gfCNCPoint5[27571] = {X 492.8890, Y 40.6660, Z -8.0000, A 0.000, B 0.000, C 0.000 }
gfCNCPoint5[27572] = {X 492.8890, Y 35.0338, Z -8.0000, A 0.000, B 0.000, C 0.000 }
gfCNCPoint5[27573] = {X 491.0677, Y 35.0338, Z -8.0000, A 0.000, B 0.000, C 0.000 }
gfCNCPoint5[27574] = {X 487.0438, Y 42.8699, Z -8.0000, A 0.000, B 0.000, C 0.000 }
gfCNCPoint5[27575] = {X 487.1809, Y 43.5111, Z -8.0000, A 0.000, B 0.000, C 0.000 }
gfCNCPoint5[27576] = {X 487.2308, Y 44.1648, Z -8.0000, A 0.000, B 0.000, C 0.000 }
gfCNCPoint5[27577] = {X 487.2310, Y 45.0000, Z -8.0000, A 0.000, B 0.000, C 0.000 }
gfCNCPoint5[27578] = {X 487.1749, Y 45.7380, Z -8.0000, A 0.000, B 0.000, C 0.000 }
gfCNCPoint5[27579] = {X 487.0078, Y 46.4590, Z -8.0000, A 0.000, B 0.000, C 0.000 }
gfCNCPoint5[27580] = {X 486.5939, Y 47.4110, Z -8.0000, A 0.000, B 0.000, C 0.000 }
gfCNCPoint5[27581] = {X 485.9879, Y 48.2538, Z -8.0000, A 0.000, B 0.000, C 0.000 }
gfCNCPoint5[27582] = {X 485.2175, Y 48.9494, Z -8.0000, A 0.000, B 0.000, C 0.000 }
gfCNCPoint5[27583] = {X 484.3173, Y 49.4663, Z -8.0000, A 0.000, B 0.000, C 0.000 }
gfCNCPoint5[27584] = {X 483.3557, Y 49.7755, Z -8.0000, A 0.000, B 0.000, C 0.000 }
gfCNCPoint5[27585] = {X 482.3510, Y 49.8800, Z -8.0000, A 0.000, B 0.000, C 0.000 }
gfCNCPoint5[27586] = {X 480.2695, Y 49.8800, Z -8.0000, A 0.000, B 0.000, C 0.000 }
gfCNCPoint5[27587] = {X 480.2695, Y 49.4000, Z -8.0000, A 0.000, B 0.000, C 0.000 }
gfCNCPoint5[27588] = {X 475.7650, Y 49.4000, Z -8.0000, A 0.000, B 0.000, C 0.000 }
gfCNCPoint5[27589] = {X 474.7859, Y 49.2897, Z -8.0000, A 0.000, B 0.000, C 0.000 }
gfCNCPoint5[27590] = {X 473.8559, Y 48.9643, Z -8.0000, A 0.000, B 0.000, C 0.000 }
gfCNCPoint5[27591] = {X 473.0216, Y 48.4401, Z -8.0000, A 0.000, B 0.000, C 0.000 }
gfCNCPoint5[27592] = {X 472.3249, Y 47.7434, Z -8.0000, A 0.000, B 0.000, C 0.000 }
gfCNCPoint5[27593] = {X 471.8007, Y 46.9091, Z -8.0000, A 0.000, B 0.000, C 0.000 }
gfCNCPoint5[27594] = {X 471.4753, Y 45.9791, Z -8.0000, A 0.000, B 0.000, C 0.000 }
gfCNCPoint5[27595] = {X 471.3650, Y 45.0000, Z -8.0000, A 0.000, B 0.000, C 0.000 }
gfCNCPoint5[27596] = {X 471.3654, Y 44.1483, Z -8.0000, A 0.000, B 0.000, C 0.000 }
gfCNCPoint5[27597] = {X 471.4638, Y 43.2816, Z -8.0000, A 0.000, B 0.000, C 0.000 }
gfCNCPoint5[27598] = {X 471.7311, Y 42.4514, Z -8.0000, A 0.000, B 0.000, C 0.000 }
gfCNCPoint5[27599] = {X 472.1570, Y 41.6903, Z -8.0000, A 0.000, B 0.000, C 0.000 }
gfCNCPoint5[27600] = {X 472.7247, Y 41.0281, Z -8.0000, A 0.000, B 0.000, C 0.000 }
gfCNCPoint5[27601] = {X 473.4118, Y 40.4909, Z -8.0000, A 0.000, B 0.000, C 0.000 }
gfCNCPoint5[27602] = {X 474.1914, Y 40.0998, Z -8.0000, A 0.000, B 0.000, C 0.000 }
gfCNCPoint5[27603] = {X 478.1276, Y 32.3951, Z -8.0000, A 0.000, B 0.000, C 0.000 }
gfCNCPoint5[27604] = {X 476.8700, Y 31.5216, Z -8.0000, A 0.000, B 0.000, C 0.000 }
gfCNCPoint5[27605] = {X 475.7393, Y 30.4892, Z -8.0000, A 0.000, B 0.000, C 0.000 }
gfCNCPoint5[27606] = {X 474.7552, Y 29.3160, Z -8.0000, A 0.000, B 0.000, C 0.000 }
gfCNCPoint5[27607] = {X 473.9353, Y 28.0229, Z -8.0000, A 0.000, B 0.000, C 0.000 }
gfCNCPoint5[27608] = {X 473.2938, Y 26.6325, Z -8.0000, A 0.000, B 0.000, C 0.000 }
gfCNCPoint5[27609] = {X 472.8423, Y 25.1695, Z -8.0000, A 0.000, B 0.000, C 0.000 }
gfCNCPoint5[27610] = {X 472.5272, Y 23.4783, Z -8.0000, A 0.000, B 0.000, C 0.000 }
gfCNCPoint5[27611] = {X 472.3864, Y 21.7639, Z -8.0000, A 0.000, B 0.000, C 0.000 }
gfCNCPoint5[27612] = {X 472.4213, Y 20.0441, Z -8.0000, A 0.000, B 0.000, C 0.000 }
gfCNCPoint5[27613] = {X 472.6315, Y 18.3368, Z -8.0000, A 0.000, B 0.000, C 0.000 }
gfCNCPoint5[27614] = {X 473.0148, Y 16.6598, Z -8.0000, A 0.000, B 0.000, C 0.000 }
gfCNCPoint5[27615] = {X 473.5615, Y 15.1345, Z -8.0000, A 0.000, B 0.000, C 0.000 }
gfCNCPoint5[27616] = {X 474.3101, Y 13.6975, Z -8.0000, A 0.000, B 0.000, C 0.000 }
gfCNCPoint5[27617] = {X 475.2468, Y 12.3754, Z -8.0000, A 0.000, B 0.000, C 0.000 }
gfCNCPoint5[27618] = {X 476.3541, Y 11.1925, Z -8.0000, A 0.000, B 0.000, C 0.000 }
gfCNCPoint5[27619] = {X 477.6116, Y 10.1708, Z -8.0000, A 0.000, B 0.000, C 0.000 }
gfCNCPoint5[27620] = {X 478.9962, Y 9.3291, Z -8.0000, A 0.000, B 0.000, C 0.000 }
gfCNCPoint5[27621] = {X 480.4821, Y 8.6830, Z -8.0000, A 0.000, B 0.000, C 0.000 }
gfCNCPoint5[27622] = {X 482.0419, Y 8.2445, Z -8.0000, A 0.000, B 0.000, C 0.000 }
gfCNCPoint5[27623] = {X 484.1468, Y 7.9165, Z -8.0000, A 0.000, B 0.000, C 0.000 }
gfCNCPoint5[27624] = {X 486.2739, Y 7.8014, Z -8.0000, A 0.000, B 0.000, C 0.000 }
gfCNCPoint5[27625] = {X 486.9707, Y 7.7892, Z -8.0000, A 0.000, B 0.000, C 0.000 }
gfCNCPoint5[27626] = {X 502.2084, Y 7.7892, Z -8.0000, A 0.000, B 0.000, C 0.000 }
gfCNCPoint5[27627] = {X 502.7400, Y 7.7934, Z -8.0000, A 0.000, B 0.000, C 0.000 }
gfCNCPoint5[27628] = {X 503.7096, Y 7.9098, Z -8.0000, A 0.000, B 0.000, C 0.000 }
gfCNCPoint5[27629] = {X 504.6294, Y 8.2380, Z -8.0000, A 0.000, B 0.000, C 0.000 }
gfCNCPoint5[27630] = {X 505.4536, Y 8.7617, Z -8.0000, A 0.000, B 0.000, C 0.000 }
gfCNCPoint5[27631] = {X 506.1415, Y 9.4549, Z -8.0000, A 0.000, B 0.000, C 0.000 }
gfCNCPoint5[27632] = {X 506.6587, Y 10.2832, Z -8.0000, A 0.000, B 0.000, C 0.000 }
gfCNCPoint5[27633] = {X 506.9797, Y 11.2055, Z -8.0000, A 0.000, B 0.000, C 0.000 }
gfCNCPoint5[27634] = {X 507.0885, Y 12.1759, Z -8.0000, A 0.000, B 0.000, C 0.000 }
gfCNCPoint5[27635] = {X 507.0883, Y 13.0233, Z -8.0000, A 0.000, B 0.000, C 0.000 }
gfCNCPoint5[27636] = {X 506.9800, Y 13.9491, Z -8.0000, A 0.000, B 0.000, C 0.000 }
gfCNCPoint5[27637] = {X 506.6792, Y 14.8313, Z -8.0000, A 0.000, B 0.000, C 0.000 }
gfCNCPoint5[27638] = {X 506.1993, Y 15.6303, Z -8.0000, A 0.000, B 0.000, C 0.000 }
gfCNCPoint5[27639] = {X 505.5618, Y 16.3103, Z -8.0000, A 0.000, B 0.000, C 0.000 }
gfCNCPoint5[27640] = {X 505.5624, Y 40.8770, Z -8.0000, A 0.000, B 0.000, C 0.000 }
gfCNCPoint5[27641] = {X 506.2064, Y 41.5660, Z -8.0000, A 0.000, B 0.000, C 0.000 }
gfCNCPoint5[27642] = {X 506.6888, Y 42.3765, Z -8.0000, A 0.000, B 0.000, C 0.000 }
gfCNCPoint5[27643] = {X 506.9874, Y 43.2711, Z -8.0000, A 0.000, B 0.000, C 0.000 }
gfCNCPoint5[27644] = {X 507.0885, Y 44.2089, Z -8.0000, A 0.000, B 0.000, C 0.000 }
gfCNCPoint5[27645] = {X 507.0885, Y 45.0000, Z -8.0000, A 0.000, B 0.000, C 0.000 }
gfCNCPoint5[27646] = {X 506.9782, Y 45.9791, Z -8.0000, A 0.000, B 0.000, C 0.000 }
gfCNCPoint5[27647] = {X 506.6528, Y 46.9091, Z -8.0000, A 0.000, B 0.000, C 0.000 }
gfCNCPoint5[27648] = {X 506.1285, Y 47.7434, Z -8.0000, A 0.000, B 0.000, C 0.000 }
gfCNCPoint5[27649] = {X 505.4318, Y 48.4401, Z -8.0000, A 0.000, B 0.000, C 0.000 }
gfCNCPoint5[27650] = {X 504.5976, Y 48.9643, Z -8.0000, A 0.000, B 0.000, C 0.000 }
gfCNCPoint5[27651] = {X 503.6676, Y 49.2897, Z -8.0000, A 0.000, B 0.000, C 0.000 }
gfCNCPoint5[27652] = {X 502.6885, Y 49.4000, Z -8.0000, A 0.000, B 0.000, C 0.000 }
gfCNCPoint5[27653] = {X 496.2450, Y 49.4000, Z -8.0000, A 0.000, B 0.000, C 0.000 }
gfCNCPoint5[27654] = {X 495.2659, Y 49.2897, Z -8.0000, A 0.000, B 0.000, C 0.000 }
gfCNCPoint5[27655] = {X 494.3359, Y 48.9643, Z -8.0000, A 0.000, B 0.000, C 0.000 }
gfCNCPoint5[27656] = {X 493.5017, Y 48.4401, Z -8.0000, A 0.000, B 0.000, C 0.000 }
gfCNCPoint5[27657] = {X 492.8050, Y 47.7433, Z -8.0000, A 0.000, B 0.000, C 0.000 }
gfCNCPoint5[27658] = {X 492.2808, Y 46.9091, Z -8.0000, A 0.000, B 0.000, C 0.000 }
gfCNCPoint5[27659] = {X 491.9553, Y 45.9791, Z -8.0000, A 0.000, B 0.000, C 0.000 }
gfCNCPoint5[27660] = {X 491.8450, Y 45.0000, Z -8.0000, A 0.000, B 0.000, C 0.000 }
gfCNCPoint5[27661] = {X 491.8454, Y 44.1483, Z -8.0000, A 0.000, B 0.000, C 0.000 }
gfCNCPoint5[27662] = {X 491.9559, Y 43.2275, Z -8.0000, A 0.000, B 0.000, C 0.000 }
gfCNCPoint5[27663] = {X 492.2568, Y 42.3503, Z -8.0000, A 0.000, B 0.000, C 0.000 }
gfCNCPoint5[27664] = {X 492.7349, Y 41.5556, Z -8.0000, A 0.000, B 0.000, C 0.000 }
gfCNCPoint5[27665] = {X 493.3690, Y 40.8789, Z -8.0000, A 0.000, B 0.000, C 0.000 }
gfCNCPoint5[27666] = {X 493.3690, Y 34.5538, Z -8.0000, A 0.000, B 0.000, C 0.000 }
gfCNCPoint5[27667] = {X 490.7746, Y 34.5538, Z -8.0000, A 0.000, B 0.000, C 0.000 }
gfCNCPoint5[27668] = {X 486.5276, Y 42.8244, Z -8.0000, A 0.000, B 0.000, C 0.000 }
gfCNCPoint5[27669] = {X 486.6948, Y 43.5077, Z -8.0000, A 0.000, B 0.000, C 0.000 }
gfCNCPoint5[27670] = {X 486.7510, Y 44.2089, Z -8.0000, A 0.000, B 0.000, C 0.000 }
gfCNCPoint5[27671] = {X 486.7510, Y 45.0000, Z -8.0000, A 0.000, B 0.000, C 0.000 }
gfCNCPoint5[27672] = {X 486.6407, Y 45.9791, Z -8.0000, A 0.000, B 0.000, C 0.000 }
gfCNCPoint5[27673] = {X 486.3153, Y 46.9091, Z -8.0000, A 0.000, B 0.000, C 0.000 }
gfCNCPoint5[27674] = {X 485.7911, Y 47.7434, Z -8.0000, A 0.000, B 0.000, C 0.000 }
gfCNCPoint5[27675] = {X 485.0944, Y 48.4401, Z -8.0000, A 0.000, B 0.000, C 0.000 }
gfCNCPoint5[27676] = {X 484.2601, Y 48.9643, Z -8.0000, A 0.000, B 0.000, C 0.000 }
gfCNCPoint5[27677] = {X 483.3301, Y 49.2897, Z -8.0000, A 0.000, B 0.000, C 0.000 }
gfCNCPoint5[27678] = {X 482.3510, Y 49.4000, Z -8.0000, A 0.000, B 0.000, C 0.000 }
gfCNCPoint5[27679] = {X 480.2695, Y 49.4000, Z -8.0000, A 0.000, B 0.000, C 0.000 }
gfCNCPoint5[27680] = {X 480.2695, Y 49.8800, Z -8.0000, A 0.000, B 0.000, C 0.000 }
gfCNCPoint5[27681] = {X 481.4067, Y 50.7435, Z -8.0000, A 0.000, B 0.000, C 0.000 }
gfCNCPoint5[27682] = {X 482.4044, Y 51.7649, Z -8.0000, A 0.000, B 0.000, C 0.000 }
gfCNCPoint5[27683] = {X 483.2411, Y 52.9219, Z -8.0000, A 0.000, B 0.000, C 0.000 }
gfCNCPoint5[27684] = {X 483.8615, Y 54.1044, Z -8.0000, A 0.000, B 0.000, C 0.000 }
gfCNCPoint5[27685] = {X 484.3133, Y 55.3610, Z -8.0000, A 0.000, B 0.000, C 0.000 }
gfCNCPoint5[27686] = {X 484.5879, Y 56.6678, Z -8.0000, A 0.000, B 0.000, C 0.000 }
gfCNCPoint5[27687] = {X 484.6800, Y 58.0000, Z -8.0000, A 0.000, B 0.000, C 0.000 }
gfCNCPoint5[27688] = {X 484.6797, Y 59.0140, Z -8.0000, A 0.000, B 0.000, C 0.000 }
gfCNCPoint5[27689] = {X 484.5593, Y 60.4582, Z -8.0000, A 0.000, B 0.000, C 0.000 }
gfCNCPoint5[27690] = {X 484.2246, Y 61.8682, Z -8.0000, A 0.000, B 0.000, C 0.000 }
gfCNCPoint5[27691] = {X 483.6832, Y 63.2124, Z -8.0000, A 0.000, B 0.000, C 0.000 }
gfCNCPoint5[27692] = {X 482.9472, Y 64.4608, Z -8.0000, A 0.000, B 0.000, C 0.000 }
gfCNCPoint5[27693] = {X 482.0330, Y 65.5853, Z -8.0000, A 0.000, B 0.000, C 0.000 }
gfCNCPoint5[27694] = {X 480.9613, Y 66.5607, Z -8.0000, A 0.000, B 0.000, C 0.000 }
gfCNCPoint5[27695] = {X 480.9617, Y 89.4449, Z -8.0000, A 0.000, B 0.000, C 0.000 }
gfCNCPoint5[27696] = {X 482.0606, Y 90.4473, Z -8.0000, A 0.000, B 0.000, C 0.000 }
gfCNCPoint5[27697] = {X 482.9926, Y 91.6066, Z -8.0000, A 0.000, B 0.000, C 0.000 }
gfCNCPoint5[27698] = {X 483.7356, Y 92.8952, Z -8.0000, A 0.000, B 0.000, C 0.000 }
gfCNCPoint5[27699] = {X 507.6811, Y 92.8952, Z -8.0000, A 0.000, B 0.000, C 0.000 }
gfCNCPoint5[27700] = {X 507.6811, Y 95.2952, Z -8.0000, A 0.000, B 0.000, C 0.000 }
gfCNCPoint5[27701] = {X 595.2967, Y 95.2952, Z -8.0000, A 0.000, B 0.000, C 0.000 }
gfCNCPoint5[27702] = {X 595.2967, Y 54.2000, Z -8.0000, A 0.000, B 0.000, C 0.000 }
gfCNCPoint5[27703] = {X 593.5565, Y 54.2000, Z -8.0000, A 0.000, B 0.000, C 0.000 }
gfCNCPoint5[27704] = {X 592.2403, Y 54.1053, Z -8.0000, A 0.000, B 0.000, C 0.000 }
gfCNCPoint5[27705] = {X 590.9511, Y 53.8233, Z -8.0000, A 0.000, B 0.000, C 0.000 }
gfCNCPoint5[27706] = {X 589.7155, Y 53.3598, Z -8.0000, A 0.000, B 0.000, C 0.000 }
gfCNCPoint5[27707] = {X 588.5589, Y 52.7242, Z -8.0000, A 0.000, B 0.000, C 0.000 }
gfCNCPoint5[27708] = {X 587.5052, Y 51.9297, Z -8.0000, A 0.000, B 0.000, C 0.000 }
gfCNCPoint5[27709] = {X 586.4956, Y 52.6955, Z -8.0000, A 0.000, B 0.000, C 0.000 }
gfCNCPoint5[27710] = {X 585.3903, Y 53.3153, Z -8.0000, A 0.000, B 0.000, C 0.000 }
gfCNCPoint5[27711] = {X 584.1375, Y 53.7999, Z -8.0000, A 0.000, B 0.000, C 0.000 }
gfCNCPoint5[27712] = {X 582.8276, Y 54.0969, Z -8.0000, A 0.000, B 0.000, C 0.000 }
gfCNCPoint5[27713] = {X 581.4884, Y 54.1999, Z -8.0000, A 0.000, B 0.000, C 0.000 }
gfCNCPoint5[27714] = {X 580.1485, Y 54.1069, Z -8.0000, A 0.000, B 0.000, C 0.000 }
gfCNCPoint5[27715] = {X 578.8364, Y 53.8198, Z -8.0000, A 0.000, B 0.000, C 0.000 }
gfCNCPoint5[27716] = {X 577.5801, Y 53.3447, Z -8.0000, A 0.000, B 0.000, C 0.000 }
gfCNCPoint5[27717] = {X 576.4063, Y 52.6917, Z -8.0000, A 0.000, B 0.000, C 0.000 }
gfCNCPoint5[27718] = {X 575.3401, Y 51.8748, Z -8.0000, A 0.000, B 0.000, C 0.000 }
gfCNCPoint5[27719] = {X 574.2798, Y 52.6879, Z -8.0000, A 0.000, B 0.000, C 0.000 }
gfCNCPoint5[27720] = {X 573.1128, Y 53.3388, Z -8.0000, A 0.000, B 0.000, C 0.000 }
gfCNCPoint5[27721] = {X 571.8638, Y 53.8139, Z -8.0000, A 0.000, B 0.000, C 0.000 }
gfCNCPoint5[27722] = {X 570.5592, Y 54.1030, Z -8.0000, A 0.000, B 0.000, C 0.000 }
gfCNCPoint5[27723] = {X 569.2264, Y 54.2000, Z -8.0000, A 0.000, B 0.000, C 0.000 }
gfCNCPoint5[27724] = {X 562.4443, Y 54.2000, Z -8.0000, A 0.000, B 0.000, C 0.000 }
gfCNCPoint5[27725] = {X 561.0051, Y 54.0867, Z -8.0000, A 0.000, B 0.000, C 0.000 }
gfCNCPoint5[27726] = {X 559.6013, Y 53.7497, Z -8.0000, A 0.000, B 0.000, C 0.000 }
gfCNCPoint5[27727] = {X 558.2676, Y 53.1973, Z -8.0000, A 0.000, B 0.000, C 0.000 }
gfCNCPoint5[27728] = {X 557.0367, Y 52.4430, Z -8.0000, A 0.000, B 0.000, C 0.000 }
gfCNCPoint5[27729] = {X 555.9389, Y 51.5054, Z -8.0000, A 0.000, B 0.000, C 0.000 }
gfCNCPoint5[27730] = {X 555.0013, Y 50.4076, Z -8.0000, A 0.000, B 0.000, C 0.000 }
gfCNCPoint5[27731] = {X 554.2470, Y 49.1767, Z -8.0000, A 0.000, B 0.000, C 0.000 }
gfCNCPoint5[27732] = {X 553.6946, Y 47.8430, Z -8.0000, A 0.000, B 0.000, C 0.000 }
gfCNCPoint5[27733] = {X 553.3576, Y 46.4392, Z -8.0000, A 0.000, B 0.000, C 0.000 }
gfCNCPoint5[27734] = {X 553.2443, Y 45.0000, Z -8.0000, A 0.000, B 0.000, C 0.000 }
gfCNCPoint5[27735] = {X 553.2443, Y 44.0496, Z -8.0000, A 0.000, B 0.000, C 0.000 }
gfCNCPoint5[27736] = {X 553.3454, Y 42.7159, Z -8.0000, A 0.000, B 0.000, C 0.000 }
gfCNCPoint5[27737] = {X 553.6383, Y 41.4109, Z -8.0000, A 0.000, B 0.000, C 0.000 }
gfCNCPoint5[27738] = {X 554.1167, Y 40.1618, Z -8.0000, A 0.000, B 0.000, C 0.000 }
gfCNCPoint5[27739] = {X 554.7706, Y 38.9951, Z -8.0000, A 0.000, B 0.000, C 0.000 }
gfCNCPoint5[27740] = {X 554.7710, Y 11.0095, Z -8.0000, A 0.000, B 0.000, C 0.000 }
gfCNCPoint5[27741] = {X 554.1213, Y 9.8543, Z -8.0000, A 0.000, B 0.000, C 0.000 }
gfCNCPoint5[27742] = {X 553.6444, Y 8.6177, Z -8.0000, A 0.000, B 0.000, C 0.000 }
gfCNCPoint5[27743] = {X 553.3501, Y 7.3255, Z -8.0000, A 0.000, B 0.000, C 0.000 }
gfCNCPoint5[27744] = {X 553.2446, Y 6.0043, Z -8.0000, A 0.000, B 0.000, C 0.000 }
gfCNCPoint5[27745] = {X 553.2443, Y 5.0000, Z -8.0000, A 0.000, B 0.000, C 0.000 }
gfCNCPoint5[27746] = {X 553.2455, Y 4.8524, Z -8.0000, A 0.000, B 0.000, C 0.000 }
gfCNCPoint5[27747] = {X 553.2490, Y 4.7048, Z -8.0000, A 0.000, B 0.000, C 0.000 }
gfCNCPoint5[27748] = {X 365.1898, Y 4.7048, Z -8.0000, A 0.000, B 0.000, C 0.000 }
gfCNCPoint5[27749] = {X 365.3286, Y 4.8536, Z -8.0000, A 0.000, B 0.000, C 0.000 }
gfCNCPoint5[27750] = {X 366.7822, Y 6.5788, Z -8.0000, A 0.000, B 0.000, C 0.000 }
gfCNCPoint5[27751] = {X 368.0909, Y 8.4164, Z -8.0000, A 0.000, B 0.000, C 0.000 }
gfCNCPoint5[27752] = {X 369.2538, Y 10.3688, Z -8.0000, A 0.000, B 0.000, C 0.000 }
gfCNCPoint5[27753] = {X 370.2531, Y 12.4098, Z -8.0000, A 0.000, B 0.000, C 0.000 }
gfCNCPoint5[27754] = {X 371.0821, Y 14.5257, Z -8.0000, A 0.000, B 0.000, C 0.000 }
gfCNCPoint5[27755] = {X 371.7352, Y 16.7024, Z -8.0000, A 0.000, B 0.000, C 0.000 }
gfCNCPoint5[27756] = {X 372.2638, Y 19.2115, Z -8.0000, A 0.000, B 0.000, C 0.000 }
gfCNCPoint5[27757] = {X 372.6048, Y 21.7529, Z -8.0000, A 0.000, B 0.000, C 0.000 }
gfCNCPoint5[27758] = {X 372.7563, Y 24.3127, Z -8.0000, A 0.000, B 0.000, C 0.000 }
gfCNCPoint5[27759] = {X 372.7176, Y 26.8766, Z -8.0000, A 0.000, B 0.000, C 0.000 }
gfCNCPoint5[27760] = {X 372.4887, Y 29.4305, Z -8.0000, A 0.000, B 0.000, C 0.000 }
gfCNCPoint5[27761] = {X 372.0711, Y 31.9605, Z -8.0000, A 0.000, B 0.000, C 0.000 }
gfCNCPoint5[27762] = {X 371.4738, Y 34.3533, Z -8.0000, A 0.000, B 0.000, C 0.000 }
gfCNCPoint5[27763] = {X 370.6645, Y 36.6830, Z -8.0000, A 0.000, B 0.000, C 0.000 }
gfCNCPoint5[27764] = {X 369.6497, Y 38.9308, Z -8.0000, A 0.000, B 0.000, C 0.000 }
gfCNCPoint5[27765] = {X 368.4377, Y 41.0787, Z -8.0000, A 0.000, B 0.000, C 0.000 }
gfCNCPoint5[27766] = {X 367.0380, Y 43.1093, Z -8.0000, A 0.000, B 0.000, C 0.000 }
gfCNCPoint5[27767] = {X 365.7250, Y 44.7116, Z -8.0000, A 0.000, B 0.000, C 0.000 }
gfCNCPoint5[27768] = {X 364.2835, Y 46.1995, Z -8.0000, A 0.000, B 0.000, C 0.000 }
gfCNCPoint5[27769] = {X 362.7235, Y 47.5626, Z -8.0000, A 0.000, B 0.000, C 0.000 }
gfCNCPoint5[27770] = {X 361.0558, Y 48.7916, Z -8.0000, A 0.000, B 0.000, C 0.000 }
gfCNCPoint5[27771] = {X 359.2919, Y 49.8780, Z -8.0000, A 0.000, B 0.000, C 0.000 }
gfCNCPoint5[27772] = {X 357.4439, Y 50.8143, Z -8.0000, A 0.000, B 0.000, C 0.000 }
gfCNCPoint5[27773] = {X 355.4662, Y 51.5800, Z -8.0000, A 0.000, B 0.000, C 0.000 }
gfCNCPoint5[27774] = {X 353.4326, Y 52.1819, Z -8.0000, A 0.000, B 0.000, C 0.000 }
gfCNCPoint5[27775] = {X 351.3566, Y 52.6160, Z -8.0000, A 0.000, B 0.000, C 0.000 }
gfCNCPoint5[27776] = {X 349.2522, Y 52.8794, Z -8.0000, A 0.000, B 0.000, C 0.000 }
gfCNCPoint5[27777] = {X 347.1334, Y 52.9702, Z -8.0000, A 0.000, B 0.000, C 0.000 }
gfCNCPoint5[27778] = {X 344.8131, Y 52.9278, Z -8.0000, A 0.000, B 0.000, C 0.000 }
gfCNCPoint5[27779] = {X 342.5052, Y 52.6847, Z -8.0000, A 0.000, B 0.000, C 0.000 }
gfCNCPoint5[27780] = {X 340.2270, Y 52.2425, Z -8.0000, A 0.000, B 0.000, C 0.000 }
gfCNCPoint5[27781] = {X 337.9957, Y 51.6048, Z -8.0000, A 0.000, B 0.000, C 0.000 }
gfCNCPoint5[27782] = {X 335.8281, Y 50.7762, Z -8.0000, A 0.000, B 0.000, C 0.000 }
gfCNCPoint5[27783] = {X 333.7403, Y 49.7629, Z -8.0000, A 0.000, B 0.000, C 0.000 }
gfCNCPoint5[27784] = {X 332.8373, Y 49.2312, Z -8.0000, A 0.000, B 0.000, C 0.000 }
gfCNCPoint5[27785] = {X 331.9559, Y 48.6646, Z -8.0000, A 0.000, B 0.000, C 0.000 }
gfCNCPoint5[27786] = {X 331.3040, Y 48.2132, Z -8.0000, A 0.000, B 0.000, C 0.000 }
gfCNCPoint5[27787] = {X 330.6657, Y 47.7427, Z -8.0000, A 0.000, B 0.000, C 0.000 }
gfCNCPoint5[27788] = {X 329.2132, Y 49.6533, Z -8.0000, A 0.000, B 0.000, C 0.000 }
gfCNCPoint5[27789] = {X 328.8701, Y 49.3884, Z -8.0000, A 0.000, B 0.000, C 0.000 }
gfCNCPoint5[27790] = {X 328.5310, Y 49.1184, Z -8.0000, A 0.000, B 0.000, C 0.000 }
gfCNCPoint5[27791] = {X 328.1263, Y 49.0389, Z -8.0000, A 0.000, B 0.000, C 0.000 }
gfCNCPoint5[27792] = {X 327.7253, Y 48.9423, Z -8.0000, A 0.000, B 0.000, C 0.000 }
gfCNCPoint5[27793] = {X 328.4844, Y 49.2660, Z -8.0000, A 0.000, B 0.000, C 0.000 }
gfCNCPoint5[27794] = {X 329.2132, Y 49.6533, Z -8.0000, A 0.000, B 0.000, C 0.000 }
gfCNCPoint5[27795] = {X 330.6657, Y 47.7427, Z -8.0000, A 0.000, B 0.000, C 0.000 }
gfCNCPoint5[27796] = {X 330.0934, Y 47.2952, Z -8.0000, A 0.000, B 0.000, C 0.000 }
gfCNCPoint5[27797] = {X 329.5333, Y 46.8324, Z -8.0000, A 0.000, B 0.000, C 0.000 }
gfCNCPoint5[27798] = {X 328.9310, Y 46.7520, Z -8.0000, A 0.000, B 0.000, C 0.000 }
gfCNCPoint5[27799] = {X 328.3374, Y 46.6216, Z -8.0000, A 0.000, B 0.000, C 0.000 }
gfCNCPoint5[27800] = {X 327.9789, Y 46.5172, Z -8.0000, A 0.000, B 0.000, C 0.000 }
gfCNCPoint5[27801] = {X 327.6263, Y 46.3944, Z -8.0000, A 0.000, B 0.000, C 0.000 }
gfCNCPoint5[27802] = {X 326.7320, Y 45.9864, Z -8.0000, A 0.000, B 0.000, C 0.000 }
gfCNCPoint5[27803] = {X 325.9009, Y 45.4616, Z -8.0000, A 0.000, B 0.000, C 0.000 }
gfCNCPoint5[27804] = {X 325.1480, Y 44.8296, Z -8.0000, A 0.000, B 0.000, C 0.000 }
gfCNCPoint5[27805] = {X 324.5140, Y 44.2115, Z -8.0000, A 0.000, B 0.000, C 0.000 }
gfCNCPoint5[27806] = {X 324.0475, Y 43.7117, Z -8.0000, A 0.000, B 0.000, C 0.000 }
gfCNCPoint5[27807] = {X 323.6300, Y 43.1703, Z -8.0000, A 0.000, B 0.000, C 0.000 }
gfCNCPoint5[27808] = {X 319.6957, Y 45.9200, Z -8.0000, A 0.000, B 0.000, C 0.000 }
gfCNCPoint5[27809] = {X 319.4780, Y 45.5976, Z -8.0000, A 0.000, B 0.000, C 0.000 }
gfCNCPoint5[27810] = {X 319.2708, Y 45.2683, Z -8.0000, A 0.000, B 0.000, C 0.000 }
gfCNCPoint5[27811] = {X 319.2514, Y 45.5948, Z -8.0000, A 0.000, B 0.000, C 0.000 }
gfCNCPoint5[27812] = {X 319.2174, Y 45.9200, Z -8.0000, A 0.000, B 0.000, C 0.000 }
gfCNCPoint5[27813] = {X 319.6957, Y 45.9200, Z -8.0000, A 0.000, B 0.000, C 0.000 }
gfCNCPoint5[27814] = {X 321.6628, Y 44.5452, Z -8.0000, A 0.000, B 0.000, C 0.000 }
gfCNCPoint5[27815] = {X 321.4884, Y 44.2868, Z -8.0000, A 0.000, B 0.000, C 0.000 }
gfCNCPoint5[27816] = {X 321.3224, Y 44.0230, Z -8.0000, A 0.000, B 0.000, C 0.000 }
gfCNCPoint5[27817] = {X 320.6707, Y 42.7444, Z -8.0000, A 0.000, B 0.000, C 0.000 }
gfCNCPoint5[27818] = {X 320.2152, Y 41.3835, Z -8.0000, A 0.000, B 0.000, C 0.000 }
gfCNCPoint5[27819] = {X 319.9659, Y 39.9703, Z -8.0000, A 0.000, B 0.000, C 0.000 }
gfCNCPoint5[27820] = {X 319.9283, Y 38.5357, Z -8.0000, A 0.000, B 0.000, C 0.000 }
gfCNCPoint5[27821] = {X 320.1032, Y 37.1113, Z -8.0000, A 0.000, B 0.000, C 0.000 }
gfCNCPoint5[27822] = {X 320.4314, Y 35.8870, Z -8.0000, A 0.000, B 0.000, C 0.000 }
gfCNCPoint5[27823] = {X 320.9167, Y 34.7161, Z -8.0000, A 0.000, B 0.000, C 0.000 }
gfCNCPoint5[27824] = {X 321.5508, Y 33.6186, Z -8.0000, A 0.000, B 0.000, C 0.000 }
gfCNCPoint5[27825] = {X 324.1393, Y 29.7483, Z -8.0000, A 0.000, B 0.000, C 0.000 }
gfCNCPoint5[27826] = {X 320.1494, Y 27.0798, Z -8.0000, A 0.000, B 0.000, C 0.000 }
gfCNCPoint5[27827] = {X 321.8041, Y 24.6058, Z -8.0000, A 0.000, B 0.000, C 0.000 }
gfCNCPoint5[27828] = {X 321.9897, Y 24.3356, Z -8.0000, A 0.000, B 0.000, C 0.000 }
gfCNCPoint5[27829] = {X 322.1814, Y 24.0697, Z -8.0000, A 0.000, B 0.000, C 0.000 }
gfCNCPoint5[27830] = {X 321.5380, Y 23.0772, Z -8.0000, A 0.000, B 0.000, C 0.000 }
gfCNCPoint5[27831] = {X 320.9778, Y 22.0356, Z -8.0000, A 0.000, B 0.000, C 0.000 }
gfCNCPoint5[27832] = {X 320.1495, Y 20.3317, Z -8.0000, A 0.000, B 0.000, C 0.000 }
gfCNCPoint5[27833] = {X 320.1494, Y 27.0798, Z -8.0000, A 0.000, B 0.000, C 0.000 }
gfCNCPoint5[27834] = {X 322.1444, Y 28.4141, Z -8.0000, A 0.000, B 0.000, C 0.000 }
gfCNCPoint5[27835] = {X 323.7974, Y 25.9425, Z -8.0000, A 0.000, B 0.000, C 0.000 }
gfCNCPoint5[27836] = {X 324.5112, Y 24.9841, Z -8.0000, A 0.000, B 0.000, C 0.000 }
gfCNCPoint5[27837] = {X 325.3162, Y 24.1010, Z -8.0000, A 0.000, B 0.000, C 0.000 }
gfCNCPoint5[27838] = {X 324.4812, Y 23.1413, Z -8.0000, A 0.000, B 0.000, C 0.000 }
gfCNCPoint5[27839] = {X 323.7518, Y 22.0991, Z -8.0000, A 0.000, B 0.000, C 0.000 }
gfCNCPoint5[27840] = {X 323.1360, Y 20.9859, Z -8.0000, A 0.000, B 0.000, C 0.000 }
gfCNCPoint5[27841] = {X 319.6151, Y 13.7428, Z -8.0000, A 0.000, B 0.000, C 0.000 }
gfCNCPoint5[27842] = {X 319.4387, Y 13.3633, Z -8.0000, A 0.000, B 0.000, C 0.000 }
gfCNCPoint5[27843] = {X 319.2755, Y 12.9779, Z -8.0000, A 0.000, B 0.000, C 0.000 }
gfCNCPoint5[27844] = {X 319.2755, Y 13.0353, Z -8.0000, A 0.000, B 0.000, C 0.000 }
gfCNCPoint5[27845] = {X 319.1699, Y 14.2150, Z -8.0000, A 0.000, B 0.000, C 0.000 }
gfCNCPoint5[27846] = {X 318.8743, Y 15.3621, Z -8.0000, A 0.000, B 0.000, C 0.000 }
gfCNCPoint5[27847] = {X 318.3966, Y 16.4460, Z -8.0000, A 0.000, B 0.000, C 0.000 }
gfCNCPoint5[27848] = {X 317.7495, Y 17.4381, Z -8.0000, A 0.000, B 0.000, C 0.000 }
gfCNCPoint5[27849] = {X 317.7493, Y 36.6430, Z -8.0000, A 0.000, B 0.000, C 0.000 }
gfCNCPoint5[27850] = {X 318.1589, Y 35.1152, Z -8.0000, A 0.000, B 0.000, C 0.000 }
gfCNCPoint5[27851] = {X 318.7645, Y 33.6540, Z -8.0000, A 0.000, B 0.000, C 0.000 }
gfCNCPoint5[27852] = {X 319.5559, Y 32.2844, Z -8.0000, A 0.000, B 0.000, C 0.000 }
gfCNCPoint5[27853] = {X 322.1444, Y 28.4141, Z -8.0000, A 0.000, B 0.000, C 0.000 }
gfCNCPoint5[27854] = {X 324.1393, Y 29.7483, Z -8.0000, A 0.000, B 0.000, C 0.000 }
gfCNCPoint5[27855] = {X 325.7907, Y 27.2791, Z -8.0000, A 0.000, B 0.000, C 0.000 }
gfCNCPoint5[27856] = {X 326.3627, Y 26.5112, Z -8.0000, A 0.000, B 0.000, C 0.000 }
gfCNCPoint5[27857] = {X 327.0077, Y 25.8035, Z -8.0000, A 0.000, B 0.000, C 0.000 }
gfCNCPoint5[27858] = {X 328.0707, Y 24.8904, Z -8.0000, A 0.000, B 0.000, C 0.000 }
gfCNCPoint5[27859] = {X 329.2543, Y 24.1403, Z -8.0000, A 0.000, B 0.000, C 0.000 }
gfCNCPoint5[27860] = {X 328.0859, Y 23.3667, Z -8.0000, A 0.000, B 0.000, C 0.000 }
gfCNCPoint5[27861] = {X 327.0414, Y 22.4326, Z -8.0000, A 0.000, B 0.000, C 0.000 }
gfCNCPoint5[27862] = {X 326.3723, Y 21.6635, Z -8.0000, A 0.000, B 0.000, C 0.000 }
gfCNCPoint5[27863] = {X 325.7878, Y 20.8284, Z -8.0000, A 0.000, B 0.000, C 0.000 }
gfCNCPoint5[27864] = {X 325.2944, Y 19.9364, Z -8.0000, A 0.000, B 0.000, C 0.000 }
gfCNCPoint5[27865] = {X 321.7736, Y 12.6936, Z -8.0000, A 0.000, B 0.000, C 0.000 }
gfCNCPoint5[27866] = {X 321.6322, Y 12.3894, Z -8.0000, A 0.000, B 0.000, C 0.000 }
gfCNCPoint5[27867] = {X 321.5015, Y 12.0806, Z -8.0000, A 0.000, B 0.000, C 0.000 }
gfCNCPoint5[27868] = {X 321.1058, Y 10.8773, Z -8.0000, A 0.000, B 0.000, C 0.000 }
gfCNCPoint5[27869] = {X 320.8706, Y 9.6327, Z -8.0000, A 0.000, B 0.000, C 0.000 }
gfCNCPoint5[27870] = {X 320.7999, Y 8.3679, Z -8.0000, A 0.000, B 0.000, C 0.000 }
gfCNCPoint5[27871] = {X 320.8950, Y 7.1048, Z -8.0000, A 0.000, B 0.000, C 0.000 }
gfCNCPoint5[27872] = {X 298.7843, Y 7.1048, Z -8.0000, A 0.000, B 0.000, C 0.000 }
gfCNCPoint5[27873] = {X 298.7843, Y 9.5048, Z -8.0000, A 0.000, B 0.000, C 0.000 }
gfCNCPoint5[27874] = {X 297.8291, Y 9.5048, Z -8.0000, A 0.000, B 0.000, C 0.000 }
gfCNCPoint5[27875] = {X 298.1371, Y 10.4754, Z -8.0000, A 0.000, B 0.000, C 0.000 }
gfCNCPoint5[27876] = {X 298.3067, Y 11.4795, Z -8.0000, A 0.000, B 0.000, C 0.000 }
gfCNCPoint5[27877] = {X 298.4763, Y 10.4754, Z -8.0000, A 0.000, B 0.000, C 0.000 }
gfCNCPoint5[27878] = {X 298.7843, Y 9.5048, Z -8.0000, A 0.000, B 0.000, C 0.000 }
gfCNCPoint5[27879] = {X 298.7843, Y 7.1048, Z -8.0000, A 0.000, B 0.000, C 0.000 }
gfCNCPoint5[27880] = {X 191.0982, Y 7.1048, Z -8.0000, A 0.000, B 0.000, C 0.000 }
gfCNCPoint5[27881] = {X 193.0709, Y 7.6380, Z -8.0000, A 0.000, B 0.000, C 0.000 }
gfCNCPoint5[27882] = {X 194.9687, Y 8.3955, Z -8.0000, A 0.000, B 0.000, C 0.000 }
gfCNCPoint5[27883] = {X 196.7663, Y 9.3672, Z -8.0000, A 0.000, B 0.000, C 0.000 }
gfCNCPoint5[27884] = {X 198.4396, Y 10.5400, Z -8.0000, A 0.000, B 0.000, C 0.000 }
gfCNCPoint5[27885] = {X 198.8609, Y 10.8896, Z -8.0000, A 0.000, B 0.000, C 0.000 }
gfCNCPoint5[27886] = {X 199.2678, Y 11.2559, Z -8.0000, A 0.000, B 0.000, C 0.000 }
gfCNCPoint5[27887] = {X 200.3530, Y 12.3983, Z -8.0000, A 0.000, B 0.000, C 0.000 }
gfCNCPoint5[27888] = {X 201.2985, Y 13.6586, Z -8.0000, A 0.000, B 0.000, C 0.000 }
gfCNCPoint5[27889] = {X 202.0918, Y 15.0200, Z -8.0000, A 0.000, B 0.000, C 0.000 }
gfCNCPoint5[27890] = {X 202.7220, Y 16.4641, Z -8.0000, A 0.000, B 0.000, C 0.000 }
gfCNCPoint5[27891] = {X 203.2157, Y 18.1838, Z -8.0000, A 0.000, B 0.000, C 0.000 }
gfCNCPoint5[27892] = {X 203.5089, Y 19.9487, Z -8.0000, A 0.000, B 0.000, C 0.000 }
gfCNCPoint5[27893] = {X 203.5980, Y 21.7356, Z -8.0000, A 0.000, B 0.000, C 0.000 }
gfCNCPoint5[27894] = {X 203.4817, Y 23.5210, Z -8.0000, A 0.000, B 0.000, C 0.000 }
gfCNCPoint5[27895] = {X 203.1614, Y 25.2812, Z -8.0000, A 0.000, B 0.000, C 0.000 }
gfCNCPoint5[27896] = {X 202.7609, Y 26.6267, Z -8.0000, A 0.000, B 0.000, C 0.000 }
gfCNCPoint5[27897] = {X 202.2092, Y 27.9175, Z -8.0000, A 0.000, B 0.000, C 0.000 }
gfCNCPoint5[27898] = {X 201.5135, Y 29.1368, Z -8.0000, A 0.000, B 0.000, C 0.000 }
gfCNCPoint5[27899] = {X 200.6829, Y 30.2686, Z -8.0000, A 0.000, B 0.000, C 0.000 }
gfCNCPoint5[27900] = {X 199.7284, Y 31.2979, Z -8.0000, A 0.000, B 0.000, C 0.000 }
gfCNCPoint5[27901] = {X 200.5674, Y 31.8704, Z -8.0000, A 0.000, B 0.000, C 0.000 }
gfCNCPoint5[27902] = {X 201.2698, Y 32.6041, Z -8.0000, A 0.000, B 0.000, C 0.000 }
gfCNCPoint5[27903] = {X 201.8050, Y 33.4673, Z -8.0000, A 0.000, B 0.000, C 0.000 }
gfCNCPoint5[27904] = {X 204.8262, Y 39.7091, Z -8.0000, A 0.000, B 0.000, C 0.000 }
gfCNCPoint5[27905] = {X 205.1508, Y 40.5847, Z -8.0000, A 0.000, B 0.000, C 0.000 }
gfCNCPoint5[27906] = {X 205.3026, Y 41.5062, Z -8.0000, A 0.000, B 0.000, C 0.000 }
gfCNCPoint5[27907] = {X 205.2761, Y 42.4397, Z -8.0000, A 0.000, B 0.000, C 0.000 }
gfCNCPoint5[27908] = {X 205.0723, Y 43.3511, Z -8.0000, A 0.000, B 0.000, C 0.000 }
gfCNCPoint5[27909] = {X 204.6986, Y 44.2070, Z -8.0000, A 0.000, B 0.000, C 0.000 }
gfCNCPoint5[27910] = {X 204.1687, Y 44.9760, Z -8.0000, A 0.000, B 0.000, C 0.000 }
gfCNCPoint5[27911] = {X 203.5020, Y 45.6299, Z -8.0000, A 0.000, B 0.000, C 0.000 }
gfCNCPoint5[27912] = {X 202.9661, Y 46.0632, Z -8.0000, A 0.000, B 0.000, C 0.000 }
gfCNCPoint5[27913] = {X 202.2143, Y 46.5644, Z -8.0000, A 0.000, B 0.000, C 0.000 }
gfCNCPoint5[27914] = {X 201.3832, Y 46.9187, Z -8.0000, A 0.000, B 0.000, C 0.000 }
gfCNCPoint5[27915] = {X 200.5010, Y 47.1139, Z -8.0000, A 0.000, B 0.000, C 0.000 }
gfCNCPoint5[27916] = {X 199.5980, Y 47.1435, Z -8.0000, A 0.000, B 0.000, C 0.000 }
gfCNCPoint5[27917] = {X 198.7050, Y 47.0063, Z -8.0000, A 0.000, B 0.000, C 0.000 }
gfCNCPoint5[27918] = {X 197.7383, Y 47.5288, Z -8.0000, A 0.000, B 0.000, C 0.000 }
gfCNCPoint5[27919] = {X 196.7525, Y 48.0143, Z -8.0000, A 0.000, B 0.000, C 0.000 }
gfCNCPoint5[27920] = {X 199.8108, Y 54.5326, Z -8.0000, A 0.000, B 0.000, C 0.000 }
gfCNCPoint5[27921] = {X 197.5975, Y 55.4825, Z -8.0000, A 0.000, B 0.000, C 0.000 }
gfCNCPoint5[27922] = {X 195.3260, Y 56.2831, Z -8.0000, A 0.000, B 0.000, C 0.000 }
gfCNCPoint5[27923] = {X 195.3577, Y 56.6291, Z -8.0000, A 0.000, B 0.000, C 0.000 }
gfCNCPoint5[27924] = {X 195.3824, Y 56.9756, Z -8.0000, A 0.000, B 0.000, C 0.000 }
gfCNCPoint5[27925] = {X 199.6721, Y 61.6585, Z -8.0000, A 0.000, B 0.000, C 0.000 }
gfCNCPoint5[27926] = {X 199.5095, Y 60.3404, Z -8.0000, A 0.000, B 0.000, C 0.000 }
gfCNCPoint5[27927] = {X 199.4510, Y 59.0136, Z -8.0000, A 0.000, B 0.000, C 0.000 }
gfCNCPoint5[27928] = {X 199.4508, Y 58.0000, Z -8.0000, A 0.000, B 0.000, C 0.000 }
gfCNCPoint5[27929] = {X 199.5410, Y 56.2570, Z -8.0000, A 0.000, B 0.000, C 0.000 }
gfCNCPoint5[27930] = {X 199.8108, Y 54.5326, Z -8.0000, A 0.000, B 0.000, C 0.000 }
gfCNCPoint5[27931] = {X 198.7914, Y 52.3598, Z -8.0000, A 0.000, B 0.000, C 0.000 }
gfCNCPoint5[27932] = {X 196.1935, Y 53.4490, Z -8.0000, A 0.000, B 0.000, C 0.000 }
gfCNCPoint5[27933] = {X 193.5138, Y 54.3181, Z -8.0000, A 0.000, B 0.000, C 0.000 }
gfCNCPoint5[27934] = {X 193.0577, Y 54.4439, Z -8.0000, A 0.000, B 0.000, C 0.000 }
gfCNCPoint5[27935] = {X 192.5994, Y 54.5619, Z -8.0000, A 0.000, B 0.000, C 0.000 }
gfCNCPoint5[27936] = {X 192.9061, Y 56.2400, Z -8.0000, A 0.000, B 0.000, C 0.000 }
gfCNCPoint5[27937] = {X 193.0134, Y 57.9425, Z -8.0000, A 0.000, B 0.000, C 0.000 }
gfCNCPoint5[27938] = {X 210.3899, Y 76.9117, Z -8.0000, A 0.000, B 0.000, C 0.000 }
gfCNCPoint5[27939] = {X 212.1596, Y 75.2906, Z -8.0000, A 0.000, B 0.000, C 0.000 }
gfCNCPoint5[27940] = {X 215.1958, Y 78.6050, Z -8.0000, A 0.000, B 0.000, C 0.000 }
gfCNCPoint5[27941] = {X 218.3251, Y 76.6004, Z -8.0000, A 0.000, B 0.000, C 0.000 }
gfCNCPoint5[27942] = {X 216.9993, Y 76.0801, Z -8.0000, A 0.000, B 0.000, C 0.000 }
gfCNCPoint5[27943] = {X 216.3731, Y 75.8859, Z -8.0000, A 0.000, B 0.000, C 0.000 }
gfCNCPoint5[27944] = {X 215.7228, Y 75.8031, Z -8.0000, A 0.000, B 0.000, C 0.000 }
gfCNCPoint5[27945] = {X 213.9275, Y 75.6421, Z -8.0000, A 0.000, B 0.000, C 0.000 }
gfCNCPoint5[27946] = {X 212.1596, Y 75.2906, Z -8.0000, A 0.000, B 0.000, C 0.000 }
gfCNCPoint5[27947] = {X 210.3899, Y 76.9117, Z -8.0000, A 0.000, B 0.000, C 0.000 }
gfCNCPoint5[27948] = {X 214.7901, Y 81.7152, Z -8.0000, A 0.000, B 0.000, C 0.000 }
gfCNCPoint5[27949] = {X 223.5800, Y 76.0842, Z -8.0000, A 0.000, B 0.000, C 0.000 }
gfCNCPoint5[27950] = {X 217.8877, Y 73.8506, Z -8.0000, A 0.000, B 0.000, C 0.000 }
gfCNCPoint5[27951] = {X 216.8696, Y 73.5378, Z -8.0000, A 0.000, B 0.000, C 0.000 }
gfCNCPoint5[27952] = {X 215.8129, Y 73.4048, Z -8.0000, A 0.000, B 0.000, C 0.000 }
gfCNCPoint5[27953] = {X 214.2710, Y 73.2668, Z -8.0000, A 0.000, B 0.000, C 0.000 }
gfCNCPoint5[27954] = {X 212.7527, Y 72.9650, Z -8.0000, A 0.000, B 0.000, C 0.000 }
gfCNCPoint5[27955] = {X 211.1542, Y 72.4571, Z -8.0000, A 0.000, B 0.000, C 0.000 }
gfCNCPoint5[27956] = {X 209.6251, Y 71.7678, Z -8.0000, A 0.000, B 0.000, C 0.000 }
gfCNCPoint5[27957] = {X 208.1860, Y 70.9062, Z -8.0000, A 0.000, B 0.000, C 0.000 }
gfCNCPoint5[27958] = {X 206.8562, Y 69.8840, Z -8.0000, A 0.000, B 0.000, C 0.000 }
gfCNCPoint5[27959] = {X 205.6535, Y 68.7149, Z -8.0000, A 0.000, B 0.000, C 0.000 }
gfCNCPoint5[27960] = {X 204.5940, Y 67.4146, Z -8.0000, A 0.000, B 0.000, C 0.000 }
gfCNCPoint5[27961] = {X 203.6921, Y 66.0004, Z -8.0000, A 0.000, B 0.000, C 0.000 }
gfCNCPoint5[27962] = {X 202.9597, Y 64.4915, Z -8.0000, A 0.000, B 0.000, C 0.000 }
gfCNCPoint5[27963] = {X 202.4068, Y 62.9080, Z -8.0000, A 0.000, B 0.000, C 0.000 }
gfCNCPoint5[27964] = {X 202.0406, Y 61.2711, Z -8.0000, A 0.000, B 0.000, C 0.000 }
gfCNCPoint5[27965] = {X 201.9013, Y 60.1430, Z -8.0000, A 0.000, B 0.000, C 0.000 }
gfCNCPoint5[27966] = {X 201.8510, Y 59.0073, Z -8.0000, A 0.000, B 0.000, C 0.000 }
gfCNCPoint5[27967] = {X 201.8508, Y 58.0000, Z -8.0000, A 0.000, B 0.000, C 0.000 }
gfCNCPoint5[27968] = {X 201.9282, Y 56.5048, Z -8.0000, A 0.000, B 0.000, C 0.000 }
gfCNCPoint5[27969] = {X 202.1596, Y 55.0256, Z -8.0000, A 0.000, B 0.000, C 0.000 }
gfCNCPoint5[27970] = {X 202.4962, Y 53.7251, Z -8.0000, A 0.000, B 0.000, C 0.000 }
gfCNCPoint5[27971] = {X 202.9519, Y 52.4615, Z -8.0000, A 0.000, B 0.000, C 0.000 }
gfCNCPoint5[27972] = {X 203.5227, Y 51.2455, Z -8.0000, A 0.000, B 0.000, C 0.000 }
gfCNCPoint5[27973] = {X 202.2636, Y 51.6571, Z -8.0000, A 0.000, B 0.000, C 0.000 }
gfCNCPoint5[27974] = {X 200.9600, Y 51.8930, Z -8.0000, A 0.000, B 0.000, C 0.000 }
gfCNCPoint5[27975] = {X 199.6365, Y 51.9489, Z -8.0000, A 0.000, B 0.000, C 0.000 }
gfCNCPoint5[27976] = {X 199.2153, Y 52.1573, Z -8.0000, A 0.000, B 0.000, C 0.000 }
gfCNCPoint5[27977] = {X 198.7914, Y 52.3598, Z -8.0000, A 0.000, B 0.000, C 0.000 }
gfCNCPoint5[27978] = {X 197.7720, Y 50.1871, Z -8.0000, A 0.000, B 0.000, C 0.000 }
gfCNCPoint5[27979] = {X 195.3553, Y 51.2001, Z -8.0000, A 0.000, B 0.000, C 0.000 }
gfCNCPoint5[27980] = {X 192.8626, Y 52.0082, Z -8.0000, A 0.000, B 0.000, C 0.000 }
gfCNCPoint5[27981] = {X 192.4426, Y 52.1241, Z -8.0000, A 0.000, B 0.000, C 0.000 }
gfCNCPoint5[27982] = {X 192.0207, Y 52.2328, Z -8.0000, A 0.000, B 0.000, C 0.000 }
gfCNCPoint5[27983] = {X 190.7206, Y 52.5198, Z -8.0000, A 0.000, B 0.000, C 0.000 }
gfCNCPoint5[27984] = {X 189.4073, Y 52.7382, Z -8.0000, A 0.000, B 0.000, C 0.000 }
gfCNCPoint5[27985] = {X 189.9009, Y 53.9123, Z -8.0000, A 0.000, B 0.000, C 0.000 }
gfCNCPoint5[27986] = {X 190.2681, Y 55.1318, Z -8.0000, A 0.000, B 0.000, C 0.000 }
gfCNCPoint5[27987] = {X 190.5268, Y 56.5555, Z -8.0000, A 0.000, B 0.000, C 0.000 }
gfCNCPoint5[27988] = {X 190.6135, Y 58.0000, Z -8.0000, A 0.000, B 0.000, C 0.000 }
gfCNCPoint5[27989] = {X 190.6132, Y 58.8754, Z -8.0000, A 0.000, B 0.000, C 0.000 }
gfCNCPoint5[27990] = {X 214.3843, Y 84.8253, Z -8.0000, A 0.000, B 0.000, C 0.000 }
gfCNCPoint5[27991] = {X 228.8348, Y 75.5681, Z -8.0000, A 0.000, B 0.000, C 0.000 }
gfCNCPoint5[27992] = {X 218.7743, Y 71.6203, Z -8.0000, A 0.000, B 0.000, C 0.000 }
gfCNCPoint5[27993] = {X 217.8425, Y 71.3060, Z -8.0000, A 0.000, B 0.000, C 0.000 }
gfCNCPoint5[27994] = {X 216.8808, Y 71.1005, Z -8.0000, A 0.000, B 0.000, C 0.000 }
gfCNCPoint5[27995] = {X 215.9020, Y 71.0065, Z -8.0000, A 0.000, B 0.000, C 0.000 }
gfCNCPoint5[27996] = {X 214.2326, Y 70.8304, Z -8.0000, A 0.000, B 0.000, C 0.000 }
gfCNCPoint5[27997] = {X 212.6037, Y 70.4247, Z -8.0000, A 0.000, B 0.000, C 0.000 }
gfCNCPoint5[27998] = {X 211.0468, Y 69.7971, Z -8.0000, A 0.000, B 0.000, C 0.000 }
gfCNCPoint5[27999] = {X 209.5920, Y 68.9598, Z -8.0000, A 0.000, B 0.000, C 0.000 }
gfCNCPoint5[28000] = {X 208.2672, Y 67.9288, Z -8.0000, A 0.000, B 0.000, C 0.000 }
gfCNCPoint5[28001] = {X 207.0982, Y 66.7241, Z -8.0000, A 0.000, B 0.000, C 0.000 }
gfCNCPoint5[28002] = {X 206.1074, Y 65.3691, Z -8.0000, A 0.000, B 0.000, C 0.000 }
gfCNCPoint5[28003] = {X 205.3141, Y 63.8897, Z -8.0000, A 0.000, B 0.000, C 0.000 }
gfCNCPoint5[28004] = {X 204.7335, Y 62.3147, Z -8.0000, A 0.000, B 0.000, C 0.000 }
gfCNCPoint5[28005] = {X 204.3768, Y 60.6744, Z -8.0000, A 0.000, B 0.000, C 0.000 }
gfCNCPoint5[28006] = {X 204.2510, Y 59.0005, Z -8.0000, A 0.000, B 0.000, C 0.000 }
gfCNCPoint5[28007] = {X 204.2508, Y 58.0000, Z -8.0000, A 0.000, B 0.000, C 0.000 }
gfCNCPoint5[28008] = {X 204.3396, Y 56.5380, Z -8.0000, A 0.000, B 0.000, C 0.000 }
gfCNCPoint5[28009] = {X 204.6047, Y 55.0975, Z -8.0000, A 0.000, B 0.000, C 0.000 }
gfCNCPoint5[28010] = {X 205.0422, Y 53.6996, Z -8.0000, A 0.000, B 0.000, C 0.000 }
gfCNCPoint5[28011] = {X 205.6456, Y 52.3650, Z -8.0000, A 0.000, B 0.000, C 0.000 }
gfCNCPoint5[28012] = {X 206.5292, Y 50.9393, Z -8.0000, A 0.000, B 0.000, C 0.000 }
gfCNCPoint5[28013] = {X 207.6017, Y 49.6496, Z -8.0000, A 0.000, B 0.000, C 0.000 }
gfCNCPoint5[28014] = {X 208.8425, Y 48.5210, Z -8.0000, A 0.000, B 0.000, C 0.000 }
gfCNCPoint5[28015] = {X 210.2277, Y 47.5751, Z -8.0000, A 0.000, B 0.000, C 0.000 }
gfCNCPoint5[28016] = {X 209.8801, Y 46.3328, Z -8.0000, A 0.000, B 0.000, C 0.000 }
gfCNCPoint5[28017] = {X 209.7572, Y 45.0487, Z -8.0000, A 0.000, B 0.000, C 0.000 }
gfCNCPoint5[28018] = {X 209.7570, Y 44.1900, Z -8.0000, A 0.000, B 0.000, C 0.000 }
gfCNCPoint5[28019] = {X 209.8558, Y 43.0016, Z -8.0000, A 0.000, B 0.000, C 0.000 }
gfCNCPoint5[28020] = {X 210.1493, Y 41.8459, Z -8.0000, A 0.000, B 0.000, C 0.000 }
gfCNCPoint5[28021] = {X 210.6296, Y 40.7544, Z -8.0000, A 0.000, B 0.000, C 0.000 }
gfCNCPoint5[28022] = {X 211.2835, Y 39.7572, Z -8.0000, A 0.000, B 0.000, C 0.000 }
gfCNCPoint5[28023] = {X 211.2835, Y 37.0741, Z -8.0000, A 0.000, B 0.000, C 0.000 }
gfCNCPoint5[28024] = {X 208.8835, Y 37.0741, Z -8.0000, A 0.000, B 0.000, C 0.000 }
gfCNCPoint5[28025] = {X 208.8835, Y 18.1956, Z -8.0000, A 0.000, B 0.000, C 0.000 }
gfCNCPoint5[28026] = {X 208.2321, Y 17.0000, Z -8.0000, A 0.000, B 0.000, C 0.000 }
gfCNCPoint5[28027] = {X 207.7549, Y 15.7248, Z -8.0000, A 0.000, B 0.000, C 0.000 }
gfCNCPoint5[28028] = {X 207.4613, Y 14.3953, Z -8.0000, A 0.000, B 0.000, C 0.000 }
gfCNCPoint5[28029] = {X 207.3572, Y 13.0378, Z -8.0000, A 0.000, B 0.000, C 0.000 }
gfCNCPoint5[28030] = {X 207.3570, Y 12.1868, Z -8.0000, A 0.000, B 0.000, C 0.000 }
gfCNCPoint5[28031] = {X 207.3580, Y 12.0458, Z -8.0000, A 0.000, B 0.000, C 0.000 }
gfCNCPoint5[28032] = {X 207.3611, Y 11.9048, Z -8.0000, A 0.000, B 0.000, C 0.000 }
gfCNCPoint5[28033] = {X 205.8585, Y 11.9048, Z -8.0000, A 0.000, B 0.000, C 0.000 }
gfCNCPoint5[28034] = {X 206.6136, Y 13.3418, Z -8.0000, A 0.000, B 0.000, C 0.000 }
gfCNCPoint5[28035] = {X 207.2390, Y 14.8398, Z -8.0000, A 0.000, B 0.000, C 0.000 }
gfCNCPoint5[28036] = {X 207.7998, Y 16.7126, Z -8.0000, A 0.000, B 0.000, C 0.000 }
gfCNCPoint5[28037] = {X 208.1786, Y 18.6305, Z -8.0000, A 0.000, B 0.000, C 0.000 }
gfCNCPoint5[28038] = {X 208.3719, Y 20.5759, Z -8.0000, A 0.000, B 0.000, C 0.000 }
gfCNCPoint5[28039] = {X 208.3779, Y 22.5309, Z -8.0000, A 0.000, B 0.000, C 0.000 }
gfCNCPoint5[28040] = {X 208.1967, Y 24.4774, Z -8.0000, A 0.000, B 0.000, C 0.000 }
gfCNCPoint5[28041] = {X 207.8298, Y 26.3977, Z -8.0000, A 0.000, B 0.000, C 0.000 }
gfCNCPoint5[28042] = {X 207.3625, Y 28.0104, Z -8.0000, A 0.000, B 0.000, C 0.000 }
gfCNCPoint5[28043] = {X 206.7389, Y 29.5694, Z -8.0000, A 0.000, B 0.000, C 0.000 }
gfCNCPoint5[28044] = {X 205.9651, Y 31.0595, Z -8.0000, A 0.000, B 0.000, C 0.000 }
gfCNCPoint5[28045] = {X 206.0467, Y 31.2170, Z -8.0000, A 0.000, B 0.000, C 0.000 }
gfCNCPoint5[28046] = {X 206.1255, Y 31.3760, Z -8.0000, A 0.000, B 0.000, C 0.000 }
gfCNCPoint5[28047] = {X 208.8835, Y 37.0741, Z -8.0000, A 0.000, B 0.000, C 0.000 }
gfCNCPoint5[28048] = {X 211.2835, Y 37.0741, Z -8.0000, A 0.000, B 0.000, C 0.000 }
gfCNCPoint5[28049] = {X 211.2833, Y 17.4381, Z -8.0000, A 0.000, B 0.000, C 0.000 }
gfCNCPoint5[28050] = {X 210.6354, Y 16.4447, Z -8.0000, A 0.000, B 0.000, C 0.000 }
gfCNCPoint5[28051] = {X 210.1574, Y 15.3592, Z -8.0000, A 0.000, B 0.000, C 0.000 }
gfCNCPoint5[28052] = {X 209.8621, Y 14.2105, Z -8.0000, A 0.000, B 0.000, C 0.000 }
gfCNCPoint5[28053] = {X 209.7572, Y 13.0291, Z -8.0000, A 0.000, B 0.000, C 0.000 }
gfCNCPoint5[28054] = {X 209.7570, Y 12.1868, Z -8.0000, A 0.000, B 0.000, C 0.000 }
gfCNCPoint5[28055] = {X 209.7578, Y 12.0808, Z -8.0000, A 0.000, B 0.000, C 0.000 }
gfCNCPoint5[28056] = {X 209.7601, Y 11.9747, Z -8.0000, A 0.000, B 0.000, C 0.000 }
gfCNCPoint5[28057] = {X 209.9068, Y 10.7176, Z -8.0000, A 0.000, B 0.000, C 0.000 }
gfCNCPoint5[28058] = {X 210.2691, Y 9.5048, Z -8.0000, A 0.000, B 0.000, C 0.000 }
gfCNCPoint5[28059] = {X 200.9091, Y 9.5048, Z -8.0000, A 0.000, B 0.000, C 0.000 }
gfCNCPoint5[28060] = {X 201.9827, Y 10.6133, Z -8.0000, A 0.000, B 0.000, C 0.000 }
gfCNCPoint5[28061] = {X 202.9444, Y 11.8200, Z -8.0000, A 0.000, B 0.000, C 0.000 }
gfCNCPoint5[28062] = {X 203.7853, Y 13.1139, Z -8.0000, A 0.000, B 0.000, C 0.000 }
gfCNCPoint5[28063] = {X 204.4387, Y 14.3566, Z -8.0000, A 0.000, B 0.000, C 0.000 }
gfCNCPoint5[28064] = {X 204.9805, Y 15.6519, Z -8.0000, A 0.000, B 0.000, C 0.000 }
gfCNCPoint5[28065] = {X 205.5529, Y 17.6384, Z -8.0000, A 0.000, B 0.000, C 0.000 }
gfCNCPoint5[28066] = {X 205.8936, Y 19.6775, Z -8.0000, A 0.000, B 0.000, C 0.000 }
gfCNCPoint5[28067] = {X 205.9980, Y 21.7422, Z -8.0000, A 0.000, B 0.000, C 0.000 }
gfCNCPoint5[28068] = {X 205.8648, Y 23.8053, Z -8.0000, A 0.000, B 0.000, C 0.000 }
gfCNCPoint5[28069] = {X 205.4956, Y 25.8394, Z -8.0000, A 0.000, B 0.000, C 0.000 }
gfCNCPoint5[28070] = {X 205.0944, Y 27.2259, Z -8.0000, A 0.000, B 0.000, C 0.000 }
gfCNCPoint5[28071] = {X 204.5587, Y 28.5661, Z -8.0000, A 0.000, B 0.000, C 0.000 }
gfCNCPoint5[28072] = {X 203.8938, Y 29.8472, Z -8.0000, A 0.000, B 0.000, C 0.000 }
gfCNCPoint5[28073] = {X 203.1061, Y 31.0567, Z -8.0000, A 0.000, B 0.000, C 0.000 }
gfCNCPoint5[28074] = {X 203.5736, Y 31.7153, Z -8.0000, A 0.000, B 0.000, C 0.000 }
gfCNCPoint5[28075] = {X 203.9653, Y 32.4217, Z -8.0000, A 0.000, B 0.000, C 0.000 }
gfCNCPoint5[28076] = {X 206.9865, Y 38.6634, Z -8.0000, A 0.000, B 0.000, C 0.000 }
gfCNCPoint5[28077] = {X 207.4240, Y 39.8017, Z -8.0000, A 0.000, B 0.000, C 0.000 }
gfCNCPoint5[28078] = {X 207.6653, Y 40.9971, Z -8.0000, A 0.000, B 0.000, C 0.000 }
gfCNCPoint5[28079] = {X 207.7038, Y 42.2159, Z -8.0000, A 0.000, B 0.000, C 0.000 }
gfCNCPoint5[28080] = {X 207.5382, Y 43.4241, Z -8.0000, A 0.000, B 0.000, C 0.000 }
gfCNCPoint5[28081] = {X 207.1733, Y 44.5877, Z -8.0000, A 0.000, B 0.000, C 0.000 }
gfCNCPoint5[28082] = {X 206.6193, Y 45.6741, Z -8.0000, A 0.000, B 0.000, C 0.000 }
gfCNCPoint5[28083] = {X 205.8917, Y 46.6527, Z -8.0000, A 0.000, B 0.000, C 0.000 }
gfCNCPoint5[28084] = {X 205.0110, Y 47.4962, Z -8.0000, A 0.000, B 0.000, C 0.000 }
gfCNCPoint5[28085] = {X 204.4756, Y 47.9291, Z -8.0000, A 0.000, B 0.000, C 0.000 }
gfCNCPoint5[28086] = {X 203.5897, Y 48.5435, Z -8.0000, A 0.000, B 0.000, C 0.000 }
gfCNCPoint5[28087] = {X 202.6229, Y 49.0206, Z -8.0000, A 0.000, B 0.000, C 0.000 }
gfCNCPoint5[28088] = {X 201.4890, Y 49.3747, Z -8.0000, A 0.000, B 0.000, C 0.000 }
gfCNCPoint5[28089] = {X 200.3127, Y 49.5400, Z -8.0000, A 0.000, B 0.000, C 0.000 }
gfCNCPoint5[28090] = {X 199.1252, Y 49.5119, Z -8.0000, A 0.000, B 0.000, C 0.000 }
gfCNCPoint5[28091] = {X 198.4526, Y 49.8577, Z -8.0000, A 0.000, B 0.000, C 0.000 }
gfCNCPoint5[28092] = {X 197.7720, Y 50.1871, Z -8.0000, A 0.000, B 0.000, C 0.000 }
gfCNCPoint5[28093] = {X 196.7525, Y 48.0143, Z -8.0000, A 0.000, B 0.000, C 0.000 }
gfCNCPoint5[28094] = {X 194.5172, Y 48.9513, Z -8.0000, A 0.000, B 0.000, C 0.000 }
gfCNCPoint5[28095] = {X 192.2113, Y 49.6982, Z -8.0000, A 0.000, B 0.000, C 0.000 }
gfCNCPoint5[28096] = {X 190.6552, Y 50.0845, Z -8.0000, A 0.000, B 0.000, C 0.000 }
gfCNCPoint5[28097] = {X 189.0758, Y 50.3612, Z -8.0000, A 0.000, B 0.000, C 0.000 }
gfCNCPoint5[28098] = {X 186.8999, Y 50.5597, Z -8.0000, A 0.000, B 0.000, C 0.000 }
gfCNCPoint5[28099] = {X 184.7149, Y 50.5506, Z -8.0000, A 0.000, B 0.000, C 0.000 }
gfCNCPoint5[28100] = {X 184.7397, Y 50.0713, Z -8.0000, A 0.000, B 0.000, C 0.000 }
gfCNCPoint5[28101] = {X 182.7590, Y 49.8805, Z -8.0000, A 0.000, B 0.000, C 0.000 }
gfCNCPoint5[28102] = {X 180.8028, Y 49.5155, Z -8.0000, A 0.000, B 0.000, C 0.000 }
gfCNCPoint5[28103] = {X 178.9541, Y 48.9787, Z -8.0000, A 0.000, B 0.000, C 0.000 }
gfCNCPoint5[28104] = {X 177.1793, Y 48.2329, Z -8.0000, A 0.000, B 0.000, C 0.000 }
gfCNCPoint5[28105] = {X 175.5021, Y 47.2879, Z -8.0000, A 0.000, B 0.000, C 0.000 }
gfCNCPoint5[28106] = {X 173.9447, Y 46.1563, Z -8.0000, A 0.000, B 0.000, C 0.000 }
gfCNCPoint5[28107] = {X 172.7965, Y 45.1084, Z -8.0000, A 0.000, B 0.000, C 0.000 }
gfCNCPoint5[28108] = {X 171.7803, Y 43.9320, Z -8.0000, A 0.000, B 0.000, C 0.000 }
gfCNCPoint5[28109] = {X 170.9106, Y 42.6435, Z -8.0000, A 0.000, B 0.000, C 0.000 }
gfCNCPoint5[28110] = {X 170.1995, Y 41.2611, Z -8.0000, A 0.000, B 0.000, C 0.000 }
gfCNCPoint5[28111] = {X 169.6571, Y 39.8043, Z -8.0000, A 0.000, B 0.000, C 0.000 }
gfCNCPoint5[28112] = {X 169.2909, Y 38.2935, Z -8.0000, A 0.000, B 0.000, C 0.000 }
gfCNCPoint5[28113] = {X 169.1804, Y 37.5992, Z -8.0000, A 0.000, B 0.000, C 0.000 }
gfCNCPoint5[28114] = {X 169.0210, Y 35.9858, Z -8.0000, A 0.000, B 0.000, C 0.000 }
gfCNCPoint5[28115] = {X 169.0381, Y 34.3646, Z -8.0000, A 0.000, B 0.000, C 0.000 }
gfCNCPoint5[28116] = {X 169.2314, Y 32.7548, Z -8.0000, A 0.000, B 0.000, C 0.000 }
gfCNCPoint5[28117] = {X 169.5987, Y 31.1757, Z -8.0000, A 0.000, B 0.000, C 0.000 }
gfCNCPoint5[28118] = {X 170.1355, Y 29.6458, Z -8.0000, A 0.000, B 0.000, C 0.000 }
gfCNCPoint5[28119] = {X 170.7622, Y 28.3583, Z -8.0000, A 0.000, B 0.000, C 0.000 }
gfCNCPoint5[28120] = {X 171.5518, Y 27.1637, Z -8.0000, A 0.000, B 0.000, C 0.000 }
gfCNCPoint5[28121] = {X 172.4908, Y 26.0826, Z -8.0000, A 0.000, B 0.000, C 0.000 }
gfCNCPoint5[28122] = {X 173.5631, Y 25.1335, Z -8.0000, A 0.000, B 0.000, C 0.000 }
gfCNCPoint5[28123] = {X 174.7502, Y 24.3326, Z -8.0000, A 0.000, B 0.000, C 0.000 }
gfCNCPoint5[28124] = {X 173.9905, Y 23.9223, Z -8.0000, A 0.000, B 0.000, C 0.000 }
gfCNCPoint5[28125] = {X 173.3255, Y 23.3715, Z -8.0000, A 0.000, B 0.000, C 0.000 }
gfCNCPoint5[28126] = {X 172.7809, Y 22.7014, Z -8.0000, A 0.000, B 0.000, C 0.000 }
gfCNCPoint5[28127] = {X 172.3776, Y 21.9378, Z -8.0000, A 0.000, B 0.000, C 0.000 }
gfCNCPoint5[28128] = {X 169.7664, Y 15.5423, Z -8.0000, A 0.000, B 0.000, C 0.000 }
gfCNCPoint5[28129] = {X 169.5125, Y 14.6752, Z -8.0000, A 0.000, B 0.000, C 0.000 }
gfCNCPoint5[28130] = {X 169.4412, Y 13.7745, Z -8.0000, A 0.000, B 0.000, C 0.000 }
gfCNCPoint5[28131] = {X 169.5553, Y 12.8782, Z -8.0000, A 0.000, B 0.000, C 0.000 }
gfCNCPoint5[28132] = {X 169.8501, Y 12.0241, Z -8.0000, A 0.000, B 0.000, C 0.000 }
gfCNCPoint5[28133] = {X 170.3131, Y 11.2482, Z -8.0000, A 0.000, B 0.000, C 0.000 }
gfCNCPoint5[28134] = {X 170.9249, Y 10.5833, Z -8.0000, A 0.000, B 0.000, C 0.000 }
gfCNCPoint5[28135] = {X 171.6596, Y 10.0573, Z -8.0000, A 0.000, B 0.000, C 0.000 }
gfCNCPoint5[28136] = {X 172.2916, Y 9.6970, Z -8.0000, A 0.000, B 0.000, C 0.000 }
gfCNCPoint5[28137] = {X 173.1772, Y 9.3227, Z -8.0000, A 0.000, B 0.000, C 0.000 }
gfCNCPoint5[28138] = {X 174.1229, Y 9.1497, Z -8.0000, A 0.000, B 0.000, C 0.000 }
gfCNCPoint5[28139] = {X 175.0836, Y 9.1862, Z -8.0000, A 0.000, B 0.000, C 0.000 }
gfCNCPoint5[28140] = {X 176.0134, Y 9.4305, Z -8.0000, A 0.000, B 0.000, C 0.000 }
gfCNCPoint5[28141] = {X 177.0960, Y 8.9703, Z -8.0000, A 0.000, B 0.000, C 0.000 }
gfCNCPoint5[28142] = {X 179.2716, Y 8.1697, Z -8.0000, A 0.000, B 0.000, C 0.000 }
gfCNCPoint5[28143] = {X 181.5154, Y 7.5873, Z -8.0000, A 0.000, B 0.000, C 0.000 }
gfCNCPoint5[28144] = {X 183.8058, Y 7.2288, Z -8.0000, A 0.000, B 0.000, C 0.000 }
gfCNCPoint5[28145] = {X 186.1203, Y 7.0978, Z -8.0000, A 0.000, B 0.000, C 0.000 }
gfCNCPoint5[28146] = {X 188.4364, Y 7.1954, Z -8.0000, A 0.000, B 0.000, C 0.000 }
gfCNCPoint5[28147] = {X 190.7317, Y 7.5208, Z -8.0000, A 0.000, B 0.000, C 0.000 }
gfCNCPoint5[28148] = {X 192.3309, Y 7.9089, Z -8.0000, A 0.000, B 0.000, C 0.000 }
gfCNCPoint5[28149] = {X 193.8855, Y 8.4482, Z -8.0000, A 0.000, B 0.000, C 0.000 }
gfCNCPoint5[28150] = {X 195.3815, Y 9.1338, Z -8.0000, A 0.000, B 0.000, C 0.000 }
gfCNCPoint5[28151] = {X 196.8050, Y 9.9594, Z -8.0000, A 0.000, B 0.000, C 0.000 }
gfCNCPoint5[28152] = {X 198.1429, Y 10.9173, Z -8.0000, A 0.000, B 0.000, C 0.000 }
gfCNCPoint5[28153] = {X 199.2097, Y 11.8667, Z -8.0000, A 0.000, B 0.000, C 0.000 }
gfCNCPoint5[28154] = {X 200.1668, Y 12.9264, Z -8.0000, A 0.000, B 0.000, C 0.000 }
gfCNCPoint5[28155] = {X 201.0030, Y 14.0840, Z -8.0000, A 0.000, B 0.000, C 0.000 }
gfCNCPoint5[28156] = {X 201.7082, Y 15.3258, Z -8.0000, A 0.000, B 0.000, C 0.000 }
gfCNCPoint5[28157] = {X 202.2741, Y 16.6369, Z -8.0000, A 0.000, B 0.000, C 0.000 }
gfCNCPoint5[28158] = {X 202.7502, Y 18.3014, Z -8.0000, A 0.000, B 0.000, C 0.000 }
gfCNCPoint5[28159] = {X 203.0328, Y 20.0095, Z -8.0000, A 0.000, B 0.000, C 0.000 }
gfCNCPoint5[28160] = {X 203.1180, Y 21.7387, Z -8.0000, A 0.000, B 0.000, C 0.000 }
gfCNCPoint5[28161] = {X 203.0048, Y 23.4663, Z -8.0000, A 0.000, B 0.000, C 0.000 }
gfCNCPoint5[28162] = {X 202.6946, Y 25.1696, Z -8.0000, A 0.000, B 0.000, C 0.000 }
gfCNCPoint5[28163] = {X 202.2598, Y 26.5986, Z -8.0000, A 0.000, B 0.000, C 0.000 }
gfCNCPoint5[28164] = {X 201.6476, Y 27.9612, Z -8.0000, A 0.000, B 0.000, C 0.000 }
gfCNCPoint5[28165] = {X 200.8678, Y 29.2352, Z -8.0000, A 0.000, B 0.000, C 0.000 }
gfCNCPoint5[28166] = {X 199.9331, Y 30.4003, Z -8.0000, A 0.000, B 0.000, C 0.000 }
gfCNCPoint5[28167] = {X 198.8583, Y 31.4377, Z -8.0000, A 0.000, B 0.000, C 0.000 }
gfCNCPoint5[28168] = {X 199.6411, Y 31.7995, Z -8.0000, A 0.000, B 0.000, C 0.000 }
gfCNCPoint5[28169] = {X 200.3382, Y 32.3071, Z -8.0000, A 0.000, B 0.000, C 0.000 }
gfCNCPoint5[28170] = {X 200.9230, Y 32.9408, Z -8.0000, A 0.000, B 0.000, C 0.000 }
gfCNCPoint5[28171] = {X 201.3730, Y 33.6764, Z -8.0000, A 0.000, B 0.000, C 0.000 }
gfCNCPoint5[28172] = {X 204.3942, Y 39.9182, Z -8.0000, A 0.000, B 0.000, C 0.000 }
gfCNCPoint5[28173] = {X 204.7207, Y 40.8441, Z -8.0000, A 0.000, B 0.000, C 0.000 }
gfCNCPoint5[28174] = {X 204.8337, Y 41.8194, Z -8.0000, A 0.000, B 0.000, C 0.000 }
gfCNCPoint5[28175] = {X 204.7276, Y 42.7955, Z -8.0000, A 0.000, B 0.000, C 0.000 }
gfCNCPoint5[28176] = {X 204.4078, Y 43.7238, Z -8.0000, A 0.000, B 0.000, C 0.000 }
gfCNCPoint5[28177] = {X 203.8900, Y 44.5580, Z -8.0000, A 0.000, B 0.000, C 0.000 }
gfCNCPoint5[28178] = {X 203.2002, Y 45.2567, Z -8.0000, A 0.000, B 0.000, C 0.000 }
gfCNCPoint5[28179] = {X 202.6643, Y 45.6900, Z -8.0000, A 0.000, B 0.000, C 0.000 }
gfCNCPoint5[28180] = {X 201.9531, Y 46.1598, Z -8.0000, A 0.000, B 0.000, C 0.000 }
gfCNCPoint5[28181] = {X 201.1648, Y 46.4840, Z -8.0000, A 0.000, B 0.000, C 0.000 }
gfCNCPoint5[28182] = {X 200.3289, Y 46.6503, Z -8.0000, A 0.000, B 0.000, C 0.000 }
gfCNCPoint5[28183] = {X 199.4766, Y 46.6527, Z -8.0000, A 0.000, B 0.000, C 0.000 }
gfCNCPoint5[28184] = {X 198.6397, Y 46.4911, Z -8.0000, A 0.000, B 0.000, C 0.000 }
gfCNCPoint5[28185] = {X 196.5324, Y 47.5874, Z -8.0000, A 0.000, B 0.000, C 0.000 }
gfCNCPoint5[28186] = {X 194.3411, Y 48.5046, Z -8.0000, A 0.000, B 0.000, C 0.000 }
gfCNCPoint5[28187] = {X 192.0811, Y 49.2362, Z -8.0000, A 0.000, B 0.000, C 0.000 }
gfCNCPoint5[28188] = {X 190.2779, Y 49.6718, Z -8.0000, A 0.000, B 0.000, C 0.000 }
gfCNCPoint5[28189] = {X 188.4449, Y 49.9573, Z -8.0000, A 0.000, B 0.000, C 0.000 }
gfCNCPoint5[28190] = {X 186.5947, Y 50.0907, Z -8.0000, A 0.000, B 0.000, C 0.000 }
gfCNCPoint5[28191] = {X 184.7397, Y 50.0713, Z -8.0000, A 0.000, B 0.000, C 0.000 }
gfCNCPoint5[28192] = {X 184.7149, Y 50.5506, Z -8.0000, A 0.000, B 0.000, C 0.000 }
gfCNCPoint5[28193] = {X 185.7101, Y 51.5039, Z -8.0000, A 0.000, B 0.000, C 0.000 }
gfCNCPoint5[28194] = {X 186.5599, Y 52.5889, Z -8.0000, A 0.000, B 0.000, C 0.000 }
gfCNCPoint5[28195] = {X 187.2470, Y 53.7836, Z -8.0000, A 0.000, B 0.000, C 0.000 }
gfCNCPoint5[28196] = {X 187.7799, Y 55.1352, Z -8.0000, A 0.000, B 0.000, C 0.000 }
gfCNCPoint5[28197] = {X 188.1045, Y 56.5513, Z -8.0000, A 0.000, B 0.000, C 0.000 }
gfCNCPoint5[28198] = {X 188.2135, Y 58.0000, Z -8.0000, A 0.000, B 0.000, C 0.000 }
gfCNCPoint5[28199] = {X 188.2132, Y 59.0140, Z -8.0000, A 0.000, B 0.000, C 0.000 }
gfCNCPoint5[28200] = {X 188.2027, Y 59.3921, Z -8.0000, A 0.000, B 0.000, C 0.000 }
gfCNCPoint5[28201] = {X 188.1774, Y 59.7694, Z -8.0000, A 0.000, B 0.000, C 0.000 }
gfCNCPoint5[28202] = {X 213.2465, Y 87.1363, Z -8.0000, A 0.000, B 0.000, C 0.000 }
gfCNCPoint5[28203] = {X 213.3837, Y 87.2837, Z -8.0000, A 0.000, B 0.000, C 0.000 }
gfCNCPoint5[28204] = {X 213.5231, Y 87.4290, Z -8.0000, A 0.000, B 0.000, C 0.000 }
gfCNCPoint5[28205] = {X 214.2174, Y 87.3788, Z -8.0000, A 0.000, B 0.000, C 0.000 }
gfCNCPoint5[28206] = {X 214.9123, Y 87.3373, Z -8.0000, A 0.000, B 0.000, C 0.000 }
gfCNCPoint5[28207] = {X 234.0897, Y 75.0520, Z -8.0000, A 0.000, B 0.000, C 0.000 }
gfCNCPoint5[28208] = {X 219.6596, Y 69.3895, Z -8.0000, A 0.000, B 0.000, C 0.000 }
gfCNCPoint5[28209] = {X 218.4690, Y 68.9892, Z -8.0000, A 0.000, B 0.000, C 0.000 }
gfCNCPoint5[28210] = {X 217.2405, Y 68.7276, Z -8.0000, A 0.000, B 0.000, C 0.000 }
gfCNCPoint5[28211] = {X 215.9902, Y 68.6081, Z -8.0000, A 0.000, B 0.000, C 0.000 }
gfCNCPoint5[28212] = {X 214.5203, Y 68.4432, Z -8.0000, A 0.000, B 0.000, C 0.000 }
gfCNCPoint5[28213] = {X 213.0926, Y 68.0564, Z -8.0000, A 0.000, B 0.000, C 0.000 }
gfCNCPoint5[28214] = {X 211.7406, Y 67.4565, Z -8.0000, A 0.000, B 0.000, C 0.000 }
gfCNCPoint5[28215] = {X 210.4957, Y 66.6577, Z -8.0000, A 0.000, B 0.000, C 0.000 }
gfCNCPoint5[28216] = {X 209.3871, Y 65.6785, Z -8.0000, A 0.000, B 0.000, C 0.000 }
gfCNCPoint5[28217] = {X 208.4406, Y 64.5419, Z -8.0000, A 0.000, B 0.000, C 0.000 }
gfCNCPoint5[28218] = {X 207.6784, Y 63.2743, Z -8.0000, A 0.000, B 0.000, C 0.000 }
gfCNCPoint5[28219] = {X 207.1181, Y 61.9054, Z -8.0000, A 0.000, B 0.000, C 0.000 }
gfCNCPoint5[28220] = {X 206.7730, Y 60.4671, Z -8.0000, A 0.000, B 0.000, C 0.000 }
gfCNCPoint5[28221] = {X 206.6510, Y 58.9930, Z -8.0000, A 0.000, B 0.000, C 0.000 }
gfCNCPoint5[28222] = {X 206.6508, Y 58.0000, Z -8.0000, A 0.000, B 0.000, C 0.000 }
gfCNCPoint5[28223] = {X 206.7577, Y 56.5655, Z -8.0000, A 0.000, B 0.000, C 0.000 }
gfCNCPoint5[28224] = {X 207.0759, Y 55.1628, Z -8.0000, A 0.000, B 0.000, C 0.000 }
gfCNCPoint5[28225] = {X 207.5986, Y 53.8226, Z -8.0000, A 0.000, B 0.000, C 0.000 }
gfCNCPoint5[28226] = {X 208.3140, Y 52.5747, Z -8.0000, A 0.000, B 0.000, C 0.000 }
gfCNCPoint5[28227] = {X 209.2065, Y 51.4466, Z -8.0000, A 0.000, B 0.000, C 0.000 }
gfCNCPoint5[28228] = {X 210.2563, Y 50.4632, Z -8.0000, A 0.000, B 0.000, C 0.000 }
gfCNCPoint5[28229] = {X 211.4402, Y 49.6463, Z -8.0000, A 0.000, B 0.000, C 0.000 }
gfCNCPoint5[28230] = {X 212.5893, Y 49.0723, Z -8.0000, A 0.000, B 0.000, C 0.000 }
gfCNCPoint5[28231] = {X 213.8042, Y 48.6556, Z -8.0000, A 0.000, B 0.000, C 0.000 }
gfCNCPoint5[28232] = {X 213.2578, Y 48.0874, Z -8.0000, A 0.000, B 0.000, C 0.000 }
gfCNCPoint5[28233] = {X 212.8100, Y 47.4386, Z -8.0000, A 0.000, B 0.000, C 0.000 }
gfCNCPoint5[28234] = {X 212.4725, Y 46.7262, Z -8.0000, A 0.000, B 0.000, C 0.000 }
gfCNCPoint5[28235] = {X 212.2401, Y 45.8965, Z -8.0000, A 0.000, B 0.000, C 0.000 }
gfCNCPoint5[28236] = {X 212.1572, Y 45.0389, Z -8.0000, A 0.000, B 0.000, C 0.000 }
gfCNCPoint5[28237] = {X 212.1570, Y 44.1900, Z -8.0000, A 0.000, B 0.000, C 0.000 }
gfCNCPoint5[28238] = {X 212.2381, Y 43.3114, Z -8.0000, A 0.000, B 0.000, C 0.000 }
gfCNCPoint5[28239] = {X 212.4787, Y 42.4624, Z -8.0000, A 0.000, B 0.000, C 0.000 }
gfCNCPoint5[28240] = {X 212.8707, Y 41.6718, Z -8.0000, A 0.000, B 0.000, C 0.000 }
gfCNCPoint5[28241] = {X 213.4008, Y 40.9664, Z -8.0000, A 0.000, B 0.000, C 0.000 }
gfCNCPoint5[28242] = {X 213.6808, Y 40.6575, Z -8.0000, A 0.000, B 0.000, C 0.000 }
gfCNCPoint5[28243] = {X 213.6835, Y 40.3041, Z -8.0000, A 0.000, B 0.000, C 0.000 }
gfCNCPoint5[28244] = {X 213.6835, Y 17.4645, Z -8.0000, A 0.000, B 0.000, C 0.000 }
gfCNCPoint5[28245] = {X 213.6782, Y 16.7695, Z -8.0000, A 0.000, B 0.000, C 0.000 }
gfCNCPoint5[28246] = {X 213.6780, Y 16.5180, Z -8.0000, A 0.000, B 0.000, C 0.000 }
gfCNCPoint5[28247] = {X 213.0394, Y 15.7768, Z -8.0000, A 0.000, B 0.000, C 0.000 }
gfCNCPoint5[28248] = {X 212.5615, Y 14.9232, Z -8.0000, A 0.000, B 0.000, C 0.000 }
gfCNCPoint5[28249] = {X 212.2634, Y 13.9914, Z -8.0000, A 0.000, B 0.000, C 0.000 }
gfCNCPoint5[28250] = {X 212.1572, Y 13.0188, Z -8.0000, A 0.000, B 0.000, C 0.000 }
gfCNCPoint5[28251] = {X 212.1570, Y 12.1868, Z -8.0000, A 0.000, B 0.000, C 0.000 }
gfCNCPoint5[28252] = {X 212.2436, Y 11.2717, Z -8.0000, A 0.000, B 0.000, C 0.000 }
gfCNCPoint5[28253] = {X 212.5002, Y 10.3890, Z -8.0000, A 0.000, B 0.000, C 0.000 }
gfCNCPoint5[28254] = {X 212.9450, Y 9.5279, Z -8.0000, A 0.000, B 0.000, C 0.000 }
gfCNCPoint5[28255] = {X 213.5511, Y 8.7718, Z -8.0000, A 0.000, B 0.000, C 0.000 }
gfCNCPoint5[28256] = {X 214.2947, Y 8.1502, Z -8.0000, A 0.000, B 0.000, C 0.000 }
gfCNCPoint5[28257] = {X 215.1464, Y 7.6879, Z -8.0000, A 0.000, B 0.000, C 0.000 }
gfCNCPoint5[28258] = {X 216.0727, Y 7.4030, Z -8.0000, A 0.000, B 0.000, C 0.000 }
gfCNCPoint5[28259] = {X 217.0370, Y 7.3068, Z -8.0000, A 0.000, B 0.000, C 0.000 }
gfCNCPoint5[28260] = {X 223.4805, Y 7.3068, Z -8.0000, A 0.000, B 0.000, C 0.000 }
gfCNCPoint5[28261] = {X 224.4448, Y 7.4030, Z -8.0000, A 0.000, B 0.000, C 0.000 }
gfCNCPoint5[28262] = {X 225.3711, Y 7.6879, Z -8.0000, A 0.000, B 0.000, C 0.000 }
gfCNCPoint5[28263] = {X 226.2228, Y 8.1502, Z -8.0000, A 0.000, B 0.000, C 0.000 }
gfCNCPoint5[28264] = {X 226.9664, Y 8.7718, Z -8.0000, A 0.000, B 0.000, C 0.000 }
gfCNCPoint5[28265] = {X 227.5725, Y 9.5279, Z -8.0000, A 0.000, B 0.000, C 0.000 }
gfCNCPoint5[28266] = {X 228.0173, Y 10.3890, Z -8.0000, A 0.000, B 0.000, C 0.000 }
gfCNCPoint5[28267] = {X 228.2739, Y 11.2717, Z -8.0000, A 0.000, B 0.000, C 0.000 }
gfCNCPoint5[28268] = {X 228.3605, Y 12.1868, Z -8.0000, A 0.000, B 0.000, C 0.000 }
gfCNCPoint5[28269] = {X 228.3603, Y 13.0237, Z -8.0000, A 0.000, B 0.000, C 0.000 }
gfCNCPoint5[28270] = {X 228.2530, Y 13.9968, Z -8.0000, A 0.000, B 0.000, C 0.000 }
gfCNCPoint5[28271] = {X 227.9536, Y 14.9288, Z -8.0000, A 0.000, B 0.000, C 0.000 }
gfCNCPoint5[28272] = {X 227.4742, Y 15.7823, Z -8.0000, A 0.000, B 0.000, C 0.000 }
gfCNCPoint5[28273] = {X 226.8342, Y 16.5230, Z -8.0000, A 0.000, B 0.000, C 0.000 }
gfCNCPoint5[28274] = {X 226.8346, Y 25.8623, Z -8.0000, A 0.000, B 0.000, C 0.000 }
gfCNCPoint5[28275] = {X 231.6346, Y 25.8620, Z -8.0000, A 0.000, B 0.000, C 0.000 }
gfCNCPoint5[28276] = {X 231.6353, Y 38.9933, Z -8.0000, A 0.000, B 0.000, C 0.000 }
gfCNCPoint5[28277] = {X 231.6440, Y 39.0069, Z -8.0000, A 0.000, B 0.000, C 0.000 }
gfCNCPoint5[28278] = {X 232.3931, Y 37.9855, Z -8.0000, A 0.000, B 0.000, C 0.000 }
gfCNCPoint5[28279] = {X 233.2692, Y 37.0706, Z -8.0000, A 0.000, B 0.000, C 0.000 }
gfCNCPoint5[28280] = {X 234.2573, Y 36.2780, Z -8.0000, A 0.000, B 0.000, C 0.000 }
gfCNCPoint5[28281] = {X 235.5689, Y 33.7107, Z -8.0000, A 0.000, B 0.000, C 0.000 }
gfCNCPoint5[28282] = {X 234.4280, Y 32.2863, Z -8.0000, A 0.000, B 0.000, C 0.000 }
gfCNCPoint5[28283] = {X 233.4495, Y 30.7459, Z -8.0000, A 0.000, B 0.000, C 0.000 }
gfCNCPoint5[28284] = {X 232.6450, Y 29.1079, Z -8.0000, A 0.000, B 0.000, C 0.000 }
gfCNCPoint5[28285] = {X 232.0243, Y 27.3918, Z -8.0000, A 0.000, B 0.000, C 0.000 }
gfCNCPoint5[28286] = {X 231.8157, Y 26.6304, Z -8.0000, A 0.000, B 0.000, C 0.000 }
gfCNCPoint5[28287] = {X 231.6346, Y 25.8620, Z -8.0000, A 0.000, B 0.000, C 0.000 }
gfCNCPoint5[28288] = {X 229.2346, Y 25.8622, Z -8.0000, A 0.000, B 0.000, C 0.000 }
gfCNCPoint5[28289] = {X 229.2353, Y 39.7501, Z -8.0000, A 0.000, B 0.000, C 0.000 }
gfCNCPoint5[28290] = {X 229.4339, Y 40.0189, Z -8.0000, A 0.000, B 0.000, C 0.000 }
gfCNCPoint5[28291] = {X 229.6200, Y 40.2966, Z -8.0000, A 0.000, B 0.000, C 0.000 }
gfCNCPoint5[28292] = {X 230.1055, Y 41.1910, Z -8.0000, A 0.000, B 0.000, C 0.000 }
gfCNCPoint5[28293] = {X 230.4616, Y 42.1443, Z -8.0000, A 0.000, B 0.000, C 0.000 }
gfCNCPoint5[28294] = {X 230.6813, Y 43.1379, Z -8.0000, A 0.000, B 0.000, C 0.000 }
gfCNCPoint5[28295] = {X 230.7603, Y 44.1524, Z -8.0000, A 0.000, B 0.000, C 0.000 }
gfCNCPoint5[28296] = {X 230.7605, Y 45.0000, Z -8.0000, A 0.000, B 0.000, C 0.000 }
gfCNCPoint5[28297] = {X 230.7459, Y 45.4609, Z -8.0000, A 0.000, B 0.000, C 0.000 }
gfCNCPoint5[28298] = {X 230.7021, Y 45.9200, Z -8.0000, A 0.000, B 0.000, C 0.000 }
gfCNCPoint5[28299] = {X 232.5859, Y 45.9200, Z -8.0000, A 0.000, B 0.000, C 0.000 }
gfCNCPoint5[28300] = {X 232.5421, Y 45.4609, Z -8.0000, A 0.000, B 0.000, C 0.000 }
gfCNCPoint5[28301] = {X 232.5275, Y 45.0000, Z -8.0000, A 0.000, B 0.000, C 0.000 }
gfCNCPoint5[28302] = {X 232.5275, Y 44.2089, Z -8.0000, A 0.000, B 0.000, C 0.000 }
gfCNCPoint5[28303] = {X 232.6006, Y 43.1798, Z -8.0000, A 0.000, B 0.000, C 0.000 }
gfCNCPoint5[28304] = {X 232.8184, Y 42.1713, Z -8.0000, A 0.000, B 0.000, C 0.000 }
gfCNCPoint5[28305] = {X 233.1766, Y 41.2038, Z -8.0000, A 0.000, B 0.000, C 0.000 }
gfCNCPoint5[28306] = {X 233.6680, Y 40.2966, Z -8.0000, A 0.000, B 0.000, C 0.000 }
gfCNCPoint5[28307] = {X 234.3527, Y 39.3876, Z -8.0000, A 0.000, B 0.000, C 0.000 }
gfCNCPoint5[28308] = {X 235.1707, Y 38.5964, Z -8.0000, A 0.000, B 0.000, C 0.000 }
gfCNCPoint5[28309] = {X 236.1021, Y 37.9424, Z -8.0000, A 0.000, B 0.000, C 0.000 }
gfCNCPoint5[28310] = {X 238.4995, Y 33.2496, Z -8.0000, A 0.000, B 0.000, C 0.000 }
gfCNCPoint5[28311] = {X 237.3856, Y 32.1417, Z -8.0000, A 0.000, B 0.000, C 0.000 }
gfCNCPoint5[28312] = {X 236.4002, Y 30.9182, Z -8.0000, A 0.000, B 0.000, C 0.000 }
gfCNCPoint5[28313] = {X 235.5551, Y 29.5938, Z -8.0000, A 0.000, B 0.000, C 0.000 }
gfCNCPoint5[28314] = {X 234.8605, Y 28.1847, Z -8.0000, A 0.000, B 0.000, C 0.000 }
gfCNCPoint5[28315] = {X 234.3248, Y 26.7078, Z -8.0000, A 0.000, B 0.000, C 0.000 }
gfCNCPoint5[28316] = {X 234.1404, Y 26.0339, Z -8.0000, A 0.000, B 0.000, C 0.000 }
gfCNCPoint5[28317] = {X 233.9802, Y 25.3538, Z -8.0000, A 0.000, B 0.000, C 0.000 }
gfCNCPoint5[28318] = {X 233.6670, Y 23.4634, Z -8.0000, A 0.000, B 0.000, C 0.000 }
gfCNCPoint5[28319] = {X 233.5408, Y 21.5513, Z -8.0000, A 0.000, B 0.000, C 0.000 }
gfCNCPoint5[28320] = {X 233.6030, Y 19.6361, Z -8.0000, A 0.000, B 0.000, C 0.000 }
gfCNCPoint5[28321] = {X 233.8529, Y 17.7362, Z -8.0000, A 0.000, B 0.000, C 0.000 }
gfCNCPoint5[28322] = {X 234.2881, Y 15.8701, Z -8.0000, A 0.000, B 0.000, C 0.000 }
gfCNCPoint5[28323] = {X 234.7344, Y 14.5414, Z -8.0000, A 0.000, B 0.000, C 0.000 }
gfCNCPoint5[28324] = {X 235.3044, Y 13.2609, Z -8.0000, A 0.000, B 0.000, C 0.000 }
gfCNCPoint5[28325] = {X 233.1605, Y 12.1823, Z -8.0000, A 0.000, B 0.000, C 0.000 }
gfCNCPoint5[28326] = {X 233.2312, Y 12.0432, Z -8.0000, A 0.000, B 0.000, C 0.000 }
gfCNCPoint5[28327] = {X 233.3032, Y 11.9048, Z -8.0000, A 0.000, B 0.000, C 0.000 }
gfCNCPoint5[28328] = {X 233.1564, Y 11.9048, Z -8.0000, A 0.000, B 0.000, C 0.000 }
gfCNCPoint5[28329] = {X 233.1594, Y 12.0435, Z -8.0000, A 0.000, B 0.000, C 0.000 }
gfCNCPoint5[28330] = {X 233.1605, Y 12.1823, Z -8.0000, A 0.000, B 0.000, C 0.000 }
gfCNCPoint5[28331] = {X 235.3044, Y 13.2609, Z -8.0000, A 0.000, B 0.000, C 0.000 }
gfCNCPoint5[28332] = {X 235.3653, Y 13.1413, Z -8.0000, A 0.000, B 0.000, C 0.000 }
gfCNCPoint5[28333] = {X 235.4273, Y 13.0221, Z -8.0000, A 0.000, B 0.000, C 0.000 }
gfCNCPoint5[28334] = {X 236.1686, Y 11.7670, Z -8.0000, A 0.000, B 0.000, C 0.000 }
gfCNCPoint5[28335] = {X 237.0298, Y 10.5907, Z -8.0000, A 0.000, B 0.000, C 0.000 }
gfCNCPoint5[28336] = {X 238.0023, Y 9.5048, Z -8.0000, A 0.000, B 0.000, C 0.000 }
gfCNCPoint5[28337] = {X 230.2484, Y 9.5048, Z -8.0000, A 0.000, B 0.000, C 0.000 }
gfCNCPoint5[28338] = {X 230.6107, Y 10.7176, Z -8.0000, A 0.000, B 0.000, C 0.000 }
gfCNCPoint5[28339] = {X 230.7574, Y 11.9747, Z -8.0000, A 0.000, B 0.000, C 0.000 }
gfCNCPoint5[28340] = {X 230.7597, Y 12.0808, Z -8.0000, A 0.000, B 0.000, C 0.000 }
gfCNCPoint5[28341] = {X 230.7605, Y 12.1868, Z -8.0000, A 0.000, B 0.000, C 0.000 }
gfCNCPoint5[28342] = {X 230.7602, Y 13.0462, Z -8.0000, A 0.000, B 0.000, C 0.000 }
gfCNCPoint5[28343] = {X 230.6532, Y 14.2231, Z -8.0000, A 0.000, B 0.000, C 0.000 }
gfCNCPoint5[28344] = {X 230.3572, Y 15.3673, Z -8.0000, A 0.000, B 0.000, C 0.000 }
gfCNCPoint5[28345] = {X 229.8801, Y 16.4484, Z -8.0000, A 0.000, B 0.000, C 0.000 }
gfCNCPoint5[28346] = {X 229.2342, Y 17.4382, Z -8.0000, A 0.000, B 0.000, C 0.000 }
gfCNCPoint5[28347] = {X 229.2346, Y 25.8622, Z -8.0000, A 0.000, B 0.000, C 0.000 }
gfCNCPoint5[28348] = {X 226.8346, Y 25.8623, Z -8.0000, A 0.000, B 0.000, C 0.000 }
gfCNCPoint5[28349] = {X 226.8354, Y 40.6649, Z -8.0000, A 0.000, B 0.000, C 0.000 }
gfCNCPoint5[28350] = {X 227.4751, Y 41.4056, Z -8.0000, A 0.000, B 0.000, C 0.000 }
gfCNCPoint5[28351] = {X 227.9541, Y 42.2591, Z -8.0000, A 0.000, B 0.000, C 0.000 }
gfCNCPoint5[28352] = {X 228.2532, Y 43.1910, Z -8.0000, A 0.000, B 0.000, C 0.000 }
gfCNCPoint5[28353] = {X 228.3603, Y 44.1638, Z -8.0000, A 0.000, B 0.000, C 0.000 }
gfCNCPoint5[28354] = {X 228.3605, Y 45.0000, Z -8.0000, A 0.000, B 0.000, C 0.000 }
gfCNCPoint5[28355] = {X 228.3507, Y 45.3090, Z -8.0000, A 0.000, B 0.000, C 0.000 }
gfCNCPoint5[28356] = {X 228.3214, Y 45.6167, Z -8.0000, A 0.000, B 0.000, C 0.000 }
gfCNCPoint5[28357] = {X 228.0910, Y 46.5992, Z -8.0000, A 0.000, B 0.000, C 0.000 }
gfCNCPoint5[28358] = {X 227.6635, Y 47.5134, Z -8.0000, A 0.000, B 0.000, C 0.000 }
gfCNCPoint5[28359] = {X 227.0571, Y 48.3200, Z -8.0000, A 0.000, B 0.000, C 0.000 }
gfCNCPoint5[28360] = {X 226.7053, Y 47.9934, Z -8.0000, A 0.000, B 0.000, C 0.000 }
gfCNCPoint5[28361] = {X 226.0261, Y 48.5889, Z -8.0000, A 0.000, B 0.000, C 0.000 }
gfCNCPoint5[28362] = {X 225.2396, Y 49.0331, Z -8.0000, A 0.000, B 0.000, C 0.000 }
gfCNCPoint5[28363] = {X 224.3790, Y 49.3073, Z -8.0000, A 0.000, B 0.000, C 0.000 }
gfCNCPoint5[28364] = {X 223.4805, Y 49.4000, Z -8.0000, A 0.000, B 0.000, C 0.000 }
gfCNCPoint5[28365] = {X 217.0370, Y 49.4000, Z -8.0000, A 0.000, B 0.000, C 0.000 }
gfCNCPoint5[28366] = {X 216.0579, Y 49.2897, Z -8.0000, A 0.000, B 0.000, C 0.000 }
gfCNCPoint5[28367] = {X 215.1279, Y 48.9643, Z -8.0000, A 0.000, B 0.000, C 0.000 }
gfCNCPoint5[28368] = {X 214.2937, Y 48.4401, Z -8.0000, A 0.000, B 0.000, C 0.000 }
gfCNCPoint5[28369] = {X 213.5970, Y 47.7433, Z -8.0000, A 0.000, B 0.000, C 0.000 }
gfCNCPoint5[28370] = {X 213.0727, Y 46.9091, Z -8.0000, A 0.000, B 0.000, C 0.000 }
gfCNCPoint5[28371] = {X 212.7473, Y 45.9791, Z -8.0000, A 0.000, B 0.000, C 0.000 }
gfCNCPoint5[28372] = {X 212.6370, Y 45.0000, Z -8.0000, A 0.000, B 0.000, C 0.000 }
gfCNCPoint5[28373] = {X 212.6370, Y 44.1900, Z -8.0000, A 0.000, B 0.000, C 0.000 }
gfCNCPoint5[28374] = {X 212.7100, Y 43.3992, Z -8.0000, A 0.000, B 0.000, C 0.000 }
gfCNCPoint5[28375] = {X 212.9266, Y 42.6352, Z -8.0000, A 0.000, B 0.000, C 0.000 }
gfCNCPoint5[28376] = {X 213.2793, Y 41.9237, Z -8.0000, A 0.000, B 0.000, C 0.000 }
gfCNCPoint5[28377] = {X 213.7564, Y 41.2888, Z -8.0000, A 0.000, B 0.000, C 0.000 }
gfCNCPoint5[28378] = {X 214.1594, Y 40.8442, Z -8.0000, A 0.000, B 0.000, C 0.000 }
gfCNCPoint5[28379] = {X 214.1635, Y 40.3060, Z -8.0000, A 0.000, B 0.000, C 0.000 }
gfCNCPoint5[28380] = {X 214.1635, Y 17.4626, Z -8.0000, A 0.000, B 0.000, C 0.000 }
gfCNCPoint5[28381] = {X 214.1582, Y 16.7691, Z -8.0000, A 0.000, B 0.000, C 0.000 }
gfCNCPoint5[28382] = {X 214.1578, Y 16.3052, Z -8.0000, A 0.000, B 0.000, C 0.000 }
gfCNCPoint5[28383] = {X 213.5159, Y 15.6166, Z -8.0000, A 0.000, B 0.000, C 0.000 }
gfCNCPoint5[28384] = {X 213.0352, Y 14.8072, Z -8.0000, A 0.000, B 0.000, C 0.000 }
gfCNCPoint5[28385] = {X 212.7377, Y 13.9140, Z -8.0000, A 0.000, B 0.000, C 0.000 }
gfCNCPoint5[28386] = {X 212.6370, Y 12.9780, Z -8.0000, A 0.000, B 0.000, C 0.000 }
gfCNCPoint5[28387] = {X 212.6370, Y 12.1868, Z -8.0000, A 0.000, B 0.000, C 0.000 }
gfCNCPoint5[28388] = {X 212.7473, Y 11.2077, Z -8.0000, A 0.000, B 0.000, C 0.000 }
gfCNCPoint5[28389] = {X 213.0728, Y 10.2777, Z -8.0000, A 0.000, B 0.000, C 0.000 }
gfCNCPoint5[28390] = {X 213.5970, Y 9.4435, Z -8.0000, A 0.000, B 0.000, C 0.000 }
gfCNCPoint5[28391] = {X 214.2937, Y 8.7468, Z -8.0000, A 0.000, B 0.000, C 0.000 }
gfCNCPoint5[28392] = {X 215.1279, Y 8.2226, Z -8.0000, A 0.000, B 0.000, C 0.000 }
gfCNCPoint5[28393] = {X 216.0579, Y 7.8971, Z -8.0000, A 0.000, B 0.000, C 0.000 }
gfCNCPoint5[28394] = {X 217.0370, Y 7.7868, Z -8.0000, A 0.000, B 0.000, C 0.000 }
gfCNCPoint5[28395] = {X 223.4805, Y 7.7868, Z -8.0000, A 0.000, B 0.000, C 0.000 }
gfCNCPoint5[28396] = {X 224.4596, Y 7.8971, Z -8.0000, A 0.000, B 0.000, C 0.000 }
gfCNCPoint5[28397] = {X 225.3896, Y 8.2226, Z -8.0000, A 0.000, B 0.000, C 0.000 }
gfCNCPoint5[28398] = {X 226.2238, Y 8.7468, Z -8.0000, A 0.000, B 0.000, C 0.000 }
gfCNCPoint5[28399] = {X 226.9205, Y 9.4435, Z -8.0000, A 0.000, B 0.000, C 0.000 }
gfCNCPoint5[28400] = {X 227.4447, Y 10.2777, Z -8.0000, A 0.000, B 0.000, C 0.000 }
gfCNCPoint5[28401] = {X 227.7702, Y 11.2077, Z -8.0000, A 0.000, B 0.000, C 0.000 }
gfCNCPoint5[28402] = {X 227.8805, Y 12.1868, Z -8.0000, A 0.000, B 0.000, C 0.000 }
gfCNCPoint5[28403] = {X 227.8802, Y 13.0233, Z -8.0000, A 0.000, B 0.000, C 0.000 }
gfCNCPoint5[28404] = {X 227.7720, Y 13.9490, Z -8.0000, A 0.000, B 0.000, C 0.000 }
gfCNCPoint5[28405] = {X 227.4713, Y 14.8310, Z -8.0000, A 0.000, B 0.000, C 0.000 }
gfCNCPoint5[28406] = {X 226.9915, Y 15.6300, Z -8.0000, A 0.000, B 0.000, C 0.000 }
gfCNCPoint5[28407] = {X 226.3542, Y 16.3100, Z -8.0000, A 0.000, B 0.000, C 0.000 }
gfCNCPoint5[28408] = {X 226.3554, Y 40.8779, Z -8.0000, A 0.000, B 0.000, C 0.000 }
gfCNCPoint5[28409] = {X 226.9990, Y 41.5668, Z -8.0000, A 0.000, B 0.000, C 0.000 }
gfCNCPoint5[28410] = {X 227.4811, Y 42.3771, Z -8.0000, A 0.000, B 0.000, C 0.000 }
gfCNCPoint5[28411] = {X 227.7795, Y 43.2715, Z -8.0000, A 0.000, B 0.000, C 0.000 }
gfCNCPoint5[28412] = {X 227.8805, Y 44.2089, Z -8.0000, A 0.000, B 0.000, C 0.000 }
gfCNCPoint5[28413] = {X 227.8805, Y 45.0000, Z -8.0000, A 0.000, B 0.000, C 0.000 }
gfCNCPoint5[28414] = {X 227.8037, Y 45.8182, Z -8.0000, A 0.000, B 0.000, C 0.000 }
gfCNCPoint5[28415] = {X 227.5762, Y 46.6079, Z -8.0000, A 0.000, B 0.000, C 0.000 }
gfCNCPoint5[28416] = {X 227.2057, Y 47.3415, Z -8.0000, A 0.000, B 0.000, C 0.000 }
gfCNCPoint5[28417] = {X 226.7053, Y 47.9934, Z -8.0000, A 0.000, B 0.000, C 0.000 }
gfCNCPoint5[28418] = {X 227.0571, Y 48.3200, Z -8.0000, A 0.000, B 0.000, C 0.000 }
gfCNCPoint5[28419] = {X 236.2309, Y 48.3200, Z -8.0000, A 0.000, B 0.000, C 0.000 }
gfCNCPoint5[28420] = {X 235.6245, Y 47.5134, Z -8.0000, A 0.000, B 0.000, C 0.000 }
gfCNCPoint5[28421] = {X 235.1970, Y 46.5992, Z -8.0000, A 0.000, B 0.000, C 0.000 }
gfCNCPoint5[28422] = {X 234.9666, Y 45.6167, Z -8.0000, A 0.000, B 0.000, C 0.000 }
gfCNCPoint5[28423] = {X 234.9373, Y 45.3090, Z -8.0000, A 0.000, B 0.000, C 0.000 }
gfCNCPoint5[28424] = {X 234.9275, Y 45.0000, Z -8.0000, A 0.000, B 0.000, C 0.000 }
gfCNCPoint5[28425] = {X 234.9275, Y 44.2089, Z -8.0000, A 0.000, B 0.000, C 0.000 }
gfCNCPoint5[28426] = {X 235.0194, Y 43.2661, Z -8.0000, A 0.000, B 0.000, C 0.000 }
gfCNCPoint5[28427] = {X 235.2918, Y 42.3588, Z -8.0000, A 0.000, B 0.000, C 0.000 }
gfCNCPoint5[28428] = {X 235.7342, Y 41.5212, Z -8.0000, A 0.000, B 0.000, C 0.000 }
gfCNCPoint5[28429] = {X 236.3302, Y 40.7849, Z -8.0000, A 0.000, B 0.000, C 0.000 }
gfCNCPoint5[28430] = {X 237.0572, Y 40.1776, Z -8.0000, A 0.000, B 0.000, C 0.000 }
gfCNCPoint5[28431] = {X 237.8878, Y 39.7222, Z -8.0000, A 0.000, B 0.000, C 0.000 }
gfCNCPoint5[28432] = {X 241.5459, Y 32.5620, Z -8.0000, A 0.000, B 0.000, C 0.000 }
gfCNCPoint5[28433] = {X 240.2113, Y 31.5590, Z -8.0000, A 0.000, B 0.000, C 0.000 }
gfCNCPoint5[28434] = {X 239.0305, Y 30.3790, Z -8.0000, A 0.000, B 0.000, C 0.000 }
gfCNCPoint5[28435] = {X 238.0266, Y 29.0451, Z -8.0000, A 0.000, B 0.000, C 0.000 }
gfCNCPoint5[28436] = {X 237.2196, Y 27.5837, Z -8.0000, A 0.000, B 0.000, C 0.000 }
gfCNCPoint5[28437] = {X 236.6253, Y 26.0236, Z -8.0000, A 0.000, B 0.000, C 0.000 }
gfCNCPoint5[28438] = {X 236.1901, Y 24.1500, Z -8.0000, A 0.000, B 0.000, C 0.000 }
gfCNCPoint5[28439] = {X 235.9682, Y 22.2394, Z -8.0000, A 0.000, B 0.000, C 0.000 }
gfCNCPoint5[28440] = {X 235.9623, Y 20.3159, Z -8.0000, A 0.000, B 0.000, C 0.000 }
gfCNCPoint5[28441] = {X 236.1725, Y 18.4039, Z -8.0000, A 0.000, B 0.000, C 0.000 }
gfCNCPoint5[28442] = {X 236.5962, Y 16.5277, Z -8.0000, A 0.000, B 0.000, C 0.000 }
gfCNCPoint5[28443] = {X 237.1156, Y 15.0570, Z -8.0000, A 0.000, B 0.000, C 0.000 }
gfCNCPoint5[28444] = {X 237.8154, Y 13.6631, Z -8.0000, A 0.000, B 0.000, C 0.000 }
gfCNCPoint5[28445] = {X 238.6845, Y 12.3680, Z -8.0000, A 0.000, B 0.000, C 0.000 }
gfCNCPoint5[28446] = {X 239.7091, Y 11.1921, Z -8.0000, A 0.000, B 0.000, C 0.000 }
gfCNCPoint5[28447] = {X 240.8736, Y 10.1536, Z -8.0000, A 0.000, B 0.000, C 0.000 }
gfCNCPoint5[28448] = {X 242.1592, Y 9.2695, Z -8.0000, A 0.000, B 0.000, C 0.000 }
gfCNCPoint5[28449] = {X 243.5455, Y 8.5536, Z -8.0000, A 0.000, B 0.000, C 0.000 }
gfCNCPoint5[28450] = {X 245.0107, Y 8.0173, Z -8.0000, A 0.000, B 0.000, C 0.000 }
gfCNCPoint5[28451] = {X 246.5316, Y 7.6691, Z -8.0000, A 0.000, B 0.000, C 0.000 }
gfCNCPoint5[28452] = {X 248.6761, Y 7.3917, Z -8.0000, A 0.000, B 0.000, C 0.000 }
gfCNCPoint5[28453] = {X 250.8369, Y 7.3092, Z -8.0000, A 0.000, B 0.000, C 0.000 }
gfCNCPoint5[28454] = {X 266.7608, Y 7.3092, Z -8.0000, A 0.000, B 0.000, C 0.000 }
gfCNCPoint5[28455] = {X 267.7192, Y 7.4107, Z -8.0000, A 0.000, B 0.000, C 0.000 }
gfCNCPoint5[28456] = {X 268.6391, Y 7.6984, Z -8.0000, A 0.000, B 0.000, C 0.000 }
gfCNCPoint5[28457] = {X 269.4845, Y 8.1612, Z -8.0000, A 0.000, B 0.000, C 0.000 }
gfCNCPoint5[28458] = {X 270.2225, Y 8.7811, Z -8.0000, A 0.000, B 0.000, C 0.000 }
gfCNCPoint5[28459] = {X 270.8244, Y 9.5339, Z -8.0000, A 0.000, B 0.000, C 0.000 }
gfCNCPoint5[28460] = {X 271.2666, Y 10.3902, Z -8.0000, A 0.000, B 0.000, C 0.000 }
gfCNCPoint5[28461] = {X 271.5236, Y 11.2718, Z -8.0000, A 0.000, B 0.000, C 0.000 }
gfCNCPoint5[28462] = {X 271.6110, Y 12.1858, Z -8.0000, A 0.000, B 0.000, C 0.000 }
gfCNCPoint5[28463] = {X 271.6108, Y 13.0237, Z -8.0000, A 0.000, B 0.000, C 0.000 }
gfCNCPoint5[28464] = {X 271.5128, Y 13.9524, Z -8.0000, A 0.000, B 0.000, C 0.000 }
gfCNCPoint5[28465] = {X 271.2396, Y 14.8453, Z -8.0000, A 0.000, B 0.000, C 0.000 }
gfCNCPoint5[28466] = {X 275.6743, Y 16.6820, Z -8.0000, A 0.000, B 0.000, C 0.000 }
gfCNCPoint5[28467] = {X 275.3129, Y 17.4561, Z -8.0000, A 0.000, B 0.000, C 0.000 }
gfCNCPoint5[28468] = {X 274.8847, Y 18.1953, Z -8.0000, A 0.000, B 0.000, C 0.000 }
gfCNCPoint5[28469] = {X 274.8850, Y 38.9920, Z -8.0000, A 0.000, B 0.000, C 0.000 }
gfCNCPoint5[28470] = {X 275.3141, Y 39.7329, Z -8.0000, A 0.000, B 0.000, C 0.000 }
gfCNCPoint5[28471] = {X 275.6760, Y 40.5088, Z -8.0000, A 0.000, B 0.000, C 0.000 }
gfCNCPoint5[28472] = {X 276.0368, Y 39.7348, Z -8.0000, A 0.000, B 0.000, C 0.000 }
gfCNCPoint5[28473] = {X 276.4641, Y 38.9954, Z -8.0000, A 0.000, B 0.000, C 0.000 }
gfCNCPoint5[28474] = {X 276.4643, Y 18.1957, Z -8.0000, A 0.000, B 0.000, C 0.000 }
gfCNCPoint5[28475] = {X 276.0359, Y 17.4563, Z -8.0000, A 0.000, B 0.000, C 0.000 }
gfCNCPoint5[28476] = {X 275.6743, Y 16.6820, Z -8.0000, A 0.000, B 0.000, C 0.000 }
gfCNCPoint5[28477] = {X 273.4570, Y 15.7637, Z -8.0000, A 0.000, B 0.000, C 0.000 }
gfCNCPoint5[28478] = {X 273.0268, Y 16.6334, Z -8.0000, A 0.000, B 0.000, C 0.000 }
gfCNCPoint5[28479] = {X 272.4847, Y 17.4383, Z -8.0000, A 0.000, B 0.000, C 0.000 }
gfCNCPoint5[28480] = {X 272.4850, Y 39.7490, Z -8.0000, A 0.000, B 0.000, C 0.000 }
gfCNCPoint5[28481] = {X 273.0277, Y 40.5550, Z -8.0000, A 0.000, B 0.000, C 0.000 }
gfCNCPoint5[28482] = {X 273.4583, Y 41.4262, Z -8.0000, A 0.000, B 0.000, C 0.000 }
gfCNCPoint5[28483] = {X 273.7587, Y 42.3086, Z -8.0000, A 0.000, B 0.000, C 0.000 }
gfCNCPoint5[28484] = {X 273.9439, Y 43.2221, Z -8.0000, A 0.000, B 0.000, C 0.000 }
gfCNCPoint5[28485] = {X 274.0108, Y 44.1519, Z -8.0000, A 0.000, B 0.000, C 0.000 }
gfCNCPoint5[28486] = {X 274.0110, Y 45.0000, Z -8.0000, A 0.000, B 0.000, C 0.000 }
gfCNCPoint5[28487] = {X 273.9884, Y 45.5734, Z -8.0000, A 0.000, B 0.000, C 0.000 }
gfCNCPoint5[28488] = {X 273.9207, Y 46.1433, Z -8.0000, A 0.000, B 0.000, C 0.000 }
gfCNCPoint5[28489] = {X 275.0713, Y 45.9760, Z -8.0000, A 0.000, B 0.000, C 0.000 }
gfCNCPoint5[28490] = {X 276.2327, Y 45.9200, Z -8.0000, A 0.000, B 0.000, C 0.000 }
gfCNCPoint5[28491] = {X 277.3960, Y 45.9200, Z -8.0000, A 0.000, B 0.000, C 0.000 }
gfCNCPoint5[28492] = {X 277.3539, Y 45.4858, Z -8.0000, A 0.000, B 0.000, C 0.000 }
gfCNCPoint5[28493] = {X 277.3378, Y 45.0498, Z -8.0000, A 0.000, B 0.000, C 0.000 }
gfCNCPoint5[28494] = {X 277.3377, Y 44.2004, Z -8.0000, A 0.000, B 0.000, C 0.000 }
gfCNCPoint5[28495] = {X 277.4023, Y 43.2542, Z -8.0000, A 0.000, B 0.000, C 0.000 }
gfCNCPoint5[28496] = {X 277.5887, Y 42.3243, Z -8.0000, A 0.000, B 0.000, C 0.000 }
gfCNCPoint5[28497] = {X 277.8938, Y 41.4262, Z -8.0000, A 0.000, B 0.000, C 0.000 }
gfCNCPoint5[28498] = {X 278.3233, Y 40.5561, Z -8.0000, A 0.000, B 0.000, C 0.000 }
gfCNCPoint5[28499] = {X 278.8641, Y 39.7503, Z -8.0000, A 0.000, B 0.000, C 0.000 }
gfCNCPoint5[28500] = {X 278.8643, Y 17.4386, Z -8.0000, A 0.000, B 0.000, C 0.000 }
gfCNCPoint5[28501] = {X 278.3220, Y 16.6336, Z -8.0000, A 0.000, B 0.000, C 0.000 }
gfCNCPoint5[28502] = {X 277.8917, Y 15.7637, Z -8.0000, A 0.000, B 0.000, C 0.000 }
gfCNCPoint5[28503] = {X 277.5902, Y 14.8788, Z -8.0000, A 0.000, B 0.000, C 0.000 }
gfCNCPoint5[28504] = {X 277.4046, Y 13.9627, Z -8.0000, A 0.000, B 0.000, C 0.000 }
gfCNCPoint5[28505] = {X 277.3379, Y 13.0303, Z -8.0000, A 0.000, B 0.000, C 0.000 }
gfCNCPoint5[28506] = {X 277.3377, Y 12.1868, Z -8.0000, A 0.000, B 0.000, C 0.000 }
gfCNCPoint5[28507] = {X 277.3952, Y 11.2737, Z -8.0000, A 0.000, B 0.000, C 0.000 }
gfCNCPoint5[28508] = {X 277.5667, Y 10.3749, Z -8.0000, A 0.000, B 0.000, C 0.000 }
gfCNCPoint5[28509] = {X 277.8497, Y 9.5048, Z -8.0000, A 0.000, B 0.000, C 0.000 }
gfCNCPoint5[28510] = {X 273.4973, Y 9.5048, Z -8.0000, A 0.000, B 0.000, C 0.000 }
gfCNCPoint5[28511] = {X 273.7805, Y 10.3737, Z -8.0000, A 0.000, B 0.000, C 0.000 }
gfCNCPoint5[28512] = {X 273.9526, Y 11.2711, Z -8.0000, A 0.000, B 0.000, C 0.000 }
gfCNCPoint5[28513] = {X 274.0110, Y 12.1831, Z -8.0000, A 0.000, B 0.000, C 0.000 }
gfCNCPoint5[28514] = {X 274.0107, Y 13.0462, Z -8.0000, A 0.000, B 0.000, C 0.000 }
gfCNCPoint5[28515] = {X 273.9427, Y 13.9732, Z -8.0000, A 0.000, B 0.000, C 0.000 }
gfCNCPoint5[28516] = {X 273.7571, Y 14.8840, Z -8.0000, A 0.000, B 0.000, C 0.000 }
gfCNCPoint5[28517] = {X 273.4570, Y 15.7637, Z -8.0000, A 0.000, B 0.000, C 0.000 }
gfCNCPoint5[28518] = {X 271.2396, Y 14.8453, Z -8.0000, A 0.000, B 0.000, C 0.000 }
gfCNCPoint5[28519] = {X 270.7507, Y 15.7451, Z -8.0000, A 0.000, B 0.000, C 0.000 }
gfCNCPoint5[28520] = {X 270.0847, Y 16.5231, Z -8.0000, A 0.000, B 0.000, C 0.000 }
gfCNCPoint5[28521] = {X 270.0851, Y 40.6641, Z -8.0000, A 0.000, B 0.000, C 0.000 }
gfCNCPoint5[28522] = {X 270.7250, Y 41.4048, Z -8.0000, A 0.000, B 0.000, C 0.000 }
gfCNCPoint5[28523] = {X 271.2043, Y 42.2583, Z -8.0000, A 0.000, B 0.000, C 0.000 }
gfCNCPoint5[28524] = {X 271.5036, Y 43.1903, Z -8.0000, A 0.000, B 0.000, C 0.000 }
gfCNCPoint5[28525] = {X 271.6108, Y 44.1633, Z -8.0000, A 0.000, B 0.000, C 0.000 }
gfCNCPoint5[28526] = {X 271.6110, Y 45.0000, Z -8.0000, A 0.000, B 0.000, C 0.000 }
gfCNCPoint5[28527] = {X 271.5959, Y 45.3844, Z -8.0000, A 0.000, B 0.000, C 0.000 }
gfCNCPoint5[28528] = {X 271.5505, Y 45.7664, Z -8.0000, A 0.000, B 0.000, C 0.000 }
gfCNCPoint5[28529] = {X 271.2989, Y 46.7171, Z -8.0000, A 0.000, B 0.000, C 0.000 }
gfCNCPoint5[28530] = {X 270.8619, Y 47.5982, Z -8.0000, A 0.000, B 0.000, C 0.000 }
gfCNCPoint5[28531] = {X 270.2571, Y 48.3736, Z -8.0000, A 0.000, B 0.000, C 0.000 }
gfCNCPoint5[28532] = {X 269.5090, Y 49.0121, Z -8.0000, A 0.000, B 0.000, C 0.000 }
gfCNCPoint5[28533] = {X 268.6482, Y 49.4876, Z -8.0000, A 0.000, B 0.000, C 0.000 }
gfCNCPoint5[28534] = {X 267.7095, Y 49.7809, Z -8.0000, A 0.000, B 0.000, C 0.000 }
gfCNCPoint5[28535] = {X 266.7310, Y 49.8800, Z -8.0000, A 0.000, B 0.000, C 0.000 }
gfCNCPoint5[28536] = {X 260.2876, Y 49.8800, Z -8.0000, A 0.000, B 0.000, C 0.000 }
gfCNCPoint5[28537] = {X 259.2646, Y 49.7716, Z -8.0000, A 0.000, B 0.000, C 0.000 }
gfCNCPoint5[28538] = {X 258.2870, Y 49.4511, Z -8.0000, A 0.000, B 0.000, C 0.000 }
gfCNCPoint5[28539] = {X 257.3984, Y 48.9328, Z -8.0000, A 0.000, B 0.000, C 0.000 }
gfCNCPoint5[28540] = {X 256.6382, Y 48.2398, Z -8.0000, A 0.000, B 0.000, C 0.000 }
gfCNCPoint5[28541] = {X 256.0401, Y 47.4028, Z -8.0000, A 0.000, B 0.000, C 0.000 }
gfCNCPoint5[28542] = {X 255.6308, Y 46.4590, Z -8.0000, A 0.000, B 0.000, C 0.000 }
gfCNCPoint5[28543] = {X 255.4666, Y 45.7568, Z -8.0000, A 0.000, B 0.000, C 0.000 }
gfCNCPoint5[28544] = {X 255.4077, Y 45.0380, Z -8.0000, A 0.000, B 0.000, C 0.000 }
gfCNCPoint5[28545] = {X 255.4080, Y 44.1417, Z -8.0000, A 0.000, B 0.000, C 0.000 }
gfCNCPoint5[28546] = {X 255.5183, Y 43.1751, Z -8.0000, A 0.000, B 0.000, C 0.000 }
gfCNCPoint5[28547] = {X 255.8181, Y 42.2497, Z -8.0000, A 0.000, B 0.000, C 0.000 }
gfCNCPoint5[28548] = {X 256.2955, Y 41.4021, Z -8.0000, A 0.000, B 0.000, C 0.000 }
gfCNCPoint5[28549] = {X 256.9315, Y 40.6660, Z -8.0000, A 0.000, B 0.000, C 0.000 }
gfCNCPoint5[28550] = {X 256.9315, Y 35.0338, Z -8.0000, A 0.000, B 0.000, C 0.000 }
gfCNCPoint5[28551] = {X 255.1109, Y 35.0338, Z -8.0000, A 0.000, B 0.000, C 0.000 }
gfCNCPoint5[28552] = {X 251.0868, Y 42.8716, Z -8.0000, A 0.000, B 0.000, C 0.000 }
gfCNCPoint5[28553] = {X 251.2237, Y 43.5133, Z -8.0000, A 0.000, B 0.000, C 0.000 }
gfCNCPoint5[28554] = {X 251.2734, Y 44.1675, Z -8.0000, A 0.000, B 0.000, C 0.000 }
gfCNCPoint5[28555] = {X 251.2736, Y 45.0000, Z -8.0000, A 0.000, B 0.000, C 0.000 }
gfCNCPoint5[28556] = {X 251.2174, Y 45.7380, Z -8.0000, A 0.000, B 0.000, C 0.000 }
gfCNCPoint5[28557] = {X 251.0503, Y 46.4590, Z -8.0000, A 0.000, B 0.000, C 0.000 }
gfCNCPoint5[28558] = {X 250.6346, Y 47.4142, Z -8.0000, A 0.000, B 0.000, C 0.000 }
gfCNCPoint5[28559] = {X 250.0255, Y 48.2593, Z -8.0000, A 0.000, B 0.000, C 0.000 }
gfCNCPoint5[28560] = {X 249.2510, Y 48.9560, Z -8.0000, A 0.000, B 0.000, C 0.000 }
gfCNCPoint5[28561] = {X 248.3462, Y 49.4723, Z -8.0000, A 0.000, B 0.000, C 0.000 }
gfCNCPoint5[28562] = {X 247.3525, Y 49.7849, Z -8.0000, A 0.000, B 0.000, C 0.000 }
gfCNCPoint5[28563] = {X 246.8754, Y 49.8562, Z -8.0000, A 0.000, B 0.000, C 0.000 }
gfCNCPoint5[28564] = {X 246.3936, Y 49.8800, Z -8.0000, A 0.000, B 0.000, C 0.000 }
gfCNCPoint5[28565] = {X 242.5312, Y 49.8800, Z -8.0000, A 0.000, B 0.000, C 0.000 }
gfCNCPoint5[28566] = {X 242.5312, Y 49.4000, Z -8.0000, A 0.000, B 0.000, C 0.000 }
gfCNCPoint5[28567] = {X 239.8075, Y 49.4000, Z -8.0000, A 0.000, B 0.000, C 0.000 }
gfCNCPoint5[28568] = {X 238.8284, Y 49.2897, Z -8.0000, A 0.000, B 0.000, C 0.000 }
gfCNCPoint5[28569] = {X 237.8984, Y 48.9643, Z -8.0000, A 0.000, B 0.000, C 0.000 }
gfCNCPoint5[28570] = {X 237.0641, Y 48.4401, Z -8.0000, A 0.000, B 0.000, C 0.000 }
gfCNCPoint5[28571] = {X 236.3674, Y 47.7434, Z -8.0000, A 0.000, B 0.000, C 0.000 }
gfCNCPoint5[28572] = {X 235.8432, Y 46.9091, Z -8.0000, A 0.000, B 0.000, C 0.000 }
gfCNCPoint5[28573] = {X 235.5178, Y 45.9791, Z -8.0000, A 0.000, B 0.000, C 0.000 }
gfCNCPoint5[28574] = {X 235.4075, Y 45.0000, Z -8.0000, A 0.000, B 0.000, C 0.000 }
gfCNCPoint5[28575] = {X 235.4079, Y 44.1483, Z -8.0000, A 0.000, B 0.000, C 0.000 }
gfCNCPoint5[28576] = {X 235.5063, Y 43.2816, Z -8.0000, A 0.000, B 0.000, C 0.000 }
gfCNCPoint5[28577] = {X 235.7737, Y 42.4514, Z -8.0000, A 0.000, B 0.000, C 0.000 }
gfCNCPoint5[28578] = {X 236.1996, Y 41.6903, Z -8.0000, A 0.000, B 0.000, C 0.000 }
gfCNCPoint5[28579] = {X 236.7672, Y 41.0281, Z -8.0000, A 0.000, B 0.000, C 0.000 }
gfCNCPoint5[28580] = {X 237.4544, Y 40.4909, Z -8.0000, A 0.000, B 0.000, C 0.000 }
gfCNCPoint5[28581] = {X 238.2339, Y 40.0998, Z -8.0000, A 0.000, B 0.000, C 0.000 }
gfCNCPoint5[28582] = {X 242.1743, Y 32.3870, Z -8.0000, A 0.000, B 0.000, C 0.000 }
gfCNCPoint5[28583] = {X 241.0106, Y 31.5943, Z -8.0000, A 0.000, B 0.000, C 0.000 }
gfCNCPoint5[28584] = {X 239.9536, Y 30.6643, Z -8.0000, A 0.000, B 0.000, C 0.000 }
gfCNCPoint5[28585] = {X 239.0191, Y 29.6111, Z -8.0000, A 0.000, B 0.000, C 0.000 }
gfCNCPoint5[28586] = {X 238.2216, Y 28.4508, Z -8.0000, A 0.000, B 0.000, C 0.000 }
gfCNCPoint5[28587] = {X 237.5731, Y 27.2011, Z -8.0000, A 0.000, B 0.000, C 0.000 }
gfCNCPoint5[28588] = {X 237.0836, Y 25.8809, Z -8.0000, A 0.000, B 0.000, C 0.000 }
gfCNCPoint5[28589] = {X 236.6618, Y 24.0613, Z -8.0000, A 0.000, B 0.000, C 0.000 }
gfCNCPoint5[28590] = {X 236.4470, Y 22.2058, Z -8.0000, A 0.000, B 0.000, C 0.000 }
gfCNCPoint5[28591] = {X 236.4418, Y 20.3379, Z -8.0000, A 0.000, B 0.000, C 0.000 }
gfCNCPoint5[28592] = {X 236.6463, Y 18.4812, Z -8.0000, A 0.000, B 0.000, C 0.000 }
gfCNCPoint5[28593] = {X 237.0579, Y 16.6592, Z -8.0000, A 0.000, B 0.000, C 0.000 }
gfCNCPoint5[28594] = {X 237.6322, Y 15.0727, Z -8.0000, A 0.000, B 0.000, C 0.000 }
gfCNCPoint5[28595] = {X 238.4247, Y 13.5832, Z -8.0000, A 0.000, B 0.000, C 0.000 }
gfCNCPoint5[28596] = {X 239.4193, Y 12.2203, Z -8.0000, A 0.000, B 0.000, C 0.000 }
gfCNCPoint5[28597] = {X 240.5962, Y 11.0113, Z -8.0000, A 0.000, B 0.000, C 0.000 }
gfCNCPoint5[28598] = {X 241.9319, Y 9.9804, Z -8.0000, A 0.000, B 0.000, C 0.000 }
gfCNCPoint5[28599] = {X 243.3996, Y 9.1483, Z -8.0000, A 0.000, B 0.000, C 0.000 }
gfCNCPoint5[28600] = {X 244.9701, Y 8.5315, Z -8.0000, A 0.000, B 0.000, C 0.000 }
gfCNCPoint5[28601] = {X 246.6118, Y 8.1424, Z -8.0000, A 0.000, B 0.000, C 0.000 }
gfCNCPoint5[28602] = {X 248.7155, Y 7.8701, Z -8.0000, A 0.000, B 0.000, C 0.000 }
gfCNCPoint5[28603] = {X 250.8352, Y 7.7892, Z -8.0000, A 0.000, B 0.000, C 0.000 }
gfCNCPoint5[28604] = {X 266.7640, Y 7.7892, Z -8.0000, A 0.000, B 0.000, C 0.000 }
gfCNCPoint5[28605] = {X 267.7371, Y 7.9061, Z -8.0000, A 0.000, B 0.000, C 0.000 }
gfCNCPoint5[28606] = {X 268.6602, Y 8.2354, Z -8.0000, A 0.000, B 0.000, C 0.000 }
gfCNCPoint5[28607] = {X 269.4876, Y 8.7608, Z -8.0000, A 0.000, B 0.000, C 0.000 }
gfCNCPoint5[28608] = {X 270.1782, Y 9.4562, Z -8.0000, A 0.000, B 0.000, C 0.000 }
gfCNCPoint5[28609] = {X 270.6979, Y 10.2872, Z -8.0000, A 0.000, B 0.000, C 0.000 }
gfCNCPoint5[28610] = {X 271.0208, Y 11.2125, Z -8.0000, A 0.000, B 0.000, C 0.000 }
gfCNCPoint5[28611] = {X 271.1310, Y 12.1864, Z -8.0000, A 0.000, B 0.000, C 0.000 }
gfCNCPoint5[28612] = {X 271.1308, Y 13.0233, Z -8.0000, A 0.000, B 0.000, C 0.000 }
gfCNCPoint5[28613] = {X 271.0226, Y 13.9490, Z -8.0000, A 0.000, B 0.000, C 0.000 }
gfCNCPoint5[28614] = {X 270.7218, Y 14.8311, Z -8.0000, A 0.000, B 0.000, C 0.000 }
gfCNCPoint5[28615] = {X 270.2420, Y 15.6300, Z -8.0000, A 0.000, B 0.000, C 0.000 }
gfCNCPoint5[28616] = {X 269.6047, Y 16.3100, Z -8.0000, A 0.000, B 0.000, C 0.000 }
gfCNCPoint5[28617] = {X 269.6051, Y 40.8771, Z -8.0000, A 0.000, B 0.000, C 0.000 }
gfCNCPoint5[28618] = {X 270.2490, Y 41.5662, Z -8.0000, A 0.000, B 0.000, C 0.000 }
gfCNCPoint5[28619] = {X 270.7314, Y 42.3766, Z -8.0000, A 0.000, B 0.000, C 0.000 }
gfCNCPoint5[28620] = {X 271.0300, Y 43.2712, Z -8.0000, A 0.000, B 0.000, C 0.000 }
gfCNCPoint5[28621] = {X 271.1310, Y 44.2089, Z -8.0000, A 0.000, B 0.000, C 0.000 }
gfCNCPoint5[28622] = {X 271.1310, Y 45.0000, Z -8.0000, A 0.000, B 0.000, C 0.000 }
gfCNCPoint5[28623] = {X 271.0207, Y 45.9791, Z -8.0000, A 0.000, B 0.000, C 0.000 }
gfCNCPoint5[28624] = {X 270.6953, Y 46.9091, Z -8.0000, A 0.000, B 0.000, C 0.000 }
gfCNCPoint5[28625] = {X 270.1711, Y 47.7434, Z -8.0000, A 0.000, B 0.000, C 0.000 }
gfCNCPoint5[28626] = {X 269.4744, Y 48.4401, Z -8.0000, A 0.000, B 0.000, C 0.000 }
gfCNCPoint5[28627] = {X 268.6401, Y 48.9643, Z -8.0000, A 0.000, B 0.000, C 0.000 }
gfCNCPoint5[28628] = {X 267.7101, Y 49.2897, Z -8.0000, A 0.000, B 0.000, C 0.000 }
gfCNCPoint5[28629] = {X 266.7310, Y 49.4000, Z -8.0000, A 0.000, B 0.000, C 0.000 }
gfCNCPoint5[28630] = {X 260.2876, Y 49.4000, Z -8.0000, A 0.000, B 0.000, C 0.000 }
gfCNCPoint5[28631] = {X 259.3085, Y 49.2897, Z -8.0000, A 0.000, B 0.000, C 0.000 }
gfCNCPoint5[28632] = {X 258.3785, Y 48.9643, Z -8.0000, A 0.000, B 0.000, C 0.000 }
gfCNCPoint5[28633] = {X 257.5442, Y 48.4401, Z -8.0000, A 0.000, B 0.000, C 0.000 }
gfCNCPoint5[28634] = {X 256.8475, Y 47.7433, Z -8.0000, A 0.000, B 0.000, C 0.000 }
gfCNCPoint5[28635] = {X 256.3233, Y 46.9091, Z -8.0000, A 0.000, B 0.000, C 0.000 }
gfCNCPoint5[28636] = {X 255.9979, Y 45.9791, Z -8.0000, A 0.000, B 0.000, C 0.000 }
gfCNCPoint5[28637] = {X 255.8876, Y 45.0000, Z -8.0000, A 0.000, B 0.000, C 0.000 }
gfCNCPoint5[28638] = {X 255.8880, Y 44.1483, Z -8.0000, A 0.000, B 0.000, C 0.000 }
gfCNCPoint5[28639] = {X 255.9984, Y 43.2275, Z -8.0000, A 0.000, B 0.000, C 0.000 }
gfCNCPoint5[28640] = {X 256.2993, Y 42.3503, Z -8.0000, A 0.000, B 0.000, C 0.000 }
gfCNCPoint5[28641] = {X 256.7775, Y 41.5556, Z -8.0000, A 0.000, B 0.000, C 0.000 }
gfCNCPoint5[28642] = {X 257.4115, Y 40.8789, Z -8.0000, A 0.000, B 0.000, C 0.000 }
gfCNCPoint5[28643] = {X 257.4115, Y 34.5538, Z -8.0000, A 0.000, B 0.000, C 0.000 }
gfCNCPoint5[28644] = {X 254.8178, Y 34.5538, Z -8.0000, A 0.000, B 0.000, C 0.000 }
gfCNCPoint5[28645] = {X 250.5706, Y 42.8260, Z -8.0000, A 0.000, B 0.000, C 0.000 }
gfCNCPoint5[28646] = {X 250.7375, Y 43.5085, Z -8.0000, A 0.000, B 0.000, C 0.000 }
gfCNCPoint5[28647] = {X 250.7936, Y 44.2089, Z -8.0000, A 0.000, B 0.000, C 0.000 }
gfCNCPoint5[28648] = {X 250.7936, Y 45.0000, Z -8.0000, A 0.000, B 0.000, C 0.000 }
gfCNCPoint5[28649] = {X 250.6832, Y 45.9791, Z -8.0000, A 0.000, B 0.000, C 0.000 }
gfCNCPoint5[28650] = {X 250.3578, Y 46.9091, Z -8.0000, A 0.000, B 0.000, C 0.000 }
gfCNCPoint5[28651] = {X 249.8336, Y 47.7434, Z -8.0000, A 0.000, B 0.000, C 0.000 }
gfCNCPoint5[28652] = {X 249.1369, Y 48.4401, Z -8.0000, A 0.000, B 0.000, C 0.000 }
gfCNCPoint5[28653] = {X 248.3026, Y 48.9643, Z -8.0000, A 0.000, B 0.000, C 0.000 }
gfCNCPoint5[28654] = {X 247.3727, Y 49.2897, Z -8.0000, A 0.000, B 0.000, C 0.000 }
gfCNCPoint5[28655] = {X 246.3936, Y 49.4000, Z -8.0000, A 0.000, B 0.000, C 0.000 }
gfCNCPoint5[28656] = {X 242.5312, Y 49.4000, Z -8.0000, A 0.000, B 0.000, C 0.000 }
gfCNCPoint5[28657] = {X 242.5312, Y 49.8800, Z -8.0000, A 0.000, B 0.000, C 0.000 }
gfCNCPoint5[28658] = {X 243.4812, Y 50.5824, Z -8.0000, A 0.000, B 0.000, C 0.000 }
gfCNCPoint5[28659] = {X 244.3384, Y 51.3953, Z -8.0000, A 0.000, B 0.000, C 0.000 }
gfCNCPoint5[28660] = {X 245.0903, Y 52.3066, Z -8.0000, A 0.000, B 0.000, C 0.000 }
gfCNCPoint5[28661] = {X 245.7256, Y 53.3027, Z -8.0000, A 0.000, B 0.000, C 0.000 }
gfCNCPoint5[28662] = {X 245.9753, Y 53.7840, Z -8.0000, A 0.000, B 0.000, C 0.000 }
gfCNCPoint5[28663] = {X 246.1977, Y 54.2785, Z -8.0000, A 0.000, B 0.000, C 0.000 }
gfCNCPoint5[28664] = {X 250.0866, Y 55.7950, Z -8.0000, A 0.000, B 0.000, C 0.000 }
gfCNCPoint5[28665] = {X 251.8777, Y 56.5059, Z -8.0000, A 0.000, B 0.000, C 0.000 }
gfCNCPoint5[28666] = {X 253.6485, Y 52.0445, Z -8.0000, A 0.000, B 0.000, C 0.000 }
gfCNCPoint5[28667] = {X 253.4928, Y 51.8945, Z -8.0000, A 0.000, B 0.000, C 0.000 }
gfCNCPoint5[28668] = {X 253.3406, Y 51.7410, Z -8.0000, A 0.000, B 0.000, C 0.000 }
gfCNCPoint5[28669] = {X 253.2765, Y 51.8064, Z -8.0000, A 0.000, B 0.000, C 0.000 }
gfCNCPoint5[28670] = {X 253.2118, Y 51.8712, Z -8.0000, A 0.000, B 0.000, C 0.000 }
gfCNCPoint5[28671] = {X 253.6485, Y 52.0445, Z -8.0000, A 0.000, B 0.000, C 0.000 }
gfCNCPoint5[28672] = {X 252.7631, Y 54.2752, Z -8.0000, A 0.000, B 0.000, C 0.000 }
gfCNCPoint5[28673] = {X 259.4029, Y 56.9107, Z -8.0000, A 0.000, B 0.000, C 0.000 }
gfCNCPoint5[28674] = {X 260.2883, Y 54.6800, Z -8.0000, A 0.000, B 0.000, C 0.000 }
gfCNCPoint5[28675] = {X 261.9958, Y 55.3577, Z -8.0000, A 0.000, B 0.000, C 0.000 }
gfCNCPoint5[28676] = {X 262.0631, Y 55.0180, Z -8.0000, A 0.000, B 0.000, C 0.000 }
gfCNCPoint5[28677] = {X 262.1384, Y 54.6800, Z -8.0000, A 0.000, B 0.000, C 0.000 }
gfCNCPoint5[28678] = {X 260.2883, Y 54.6800, Z -8.0000, A 0.000, B 0.000, C 0.000 }
gfCNCPoint5[28679] = {X 259.4029, Y 56.9107, Z -8.0000, A 0.000, B 0.000, C 0.000 }
gfCNCPoint5[28680] = {X 264.1528, Y 58.7960, Z -8.0000, A 0.000, B 0.000, C 0.000 }
gfCNCPoint5[28681] = {X 264.1527, Y 58.0000, Z -8.0000, A 0.000, B 0.000, C 0.000 }
gfCNCPoint5[28682] = {X 264.2035, Y 56.8932, Z -8.0000, A 0.000, B 0.000, C 0.000 }
gfCNCPoint5[28683] = {X 264.3555, Y 55.7957, Z -8.0000, A 0.000, B 0.000, C 0.000 }
gfCNCPoint5[28684] = {X 264.4116, Y 55.5123, Z -8.0000, A 0.000, B 0.000, C 0.000 }
gfCNCPoint5[28685] = {X 264.4745, Y 55.2303, Z -8.0000, A 0.000, B 0.000, C 0.000 }
gfCNCPoint5[28686] = {X 264.9369, Y 53.7185, Z -8.0000, A 0.000, B 0.000, C 0.000 }
gfCNCPoint5[28687] = {X 265.5928, Y 52.2800, Z -8.0000, A 0.000, B 0.000, C 0.000 }
gfCNCPoint5[28688] = {X 260.2876, Y 52.2800, Z -8.0000, A 0.000, B 0.000, C 0.000 }
gfCNCPoint5[28689] = {X 259.1913, Y 52.1970, Z -8.0000, A 0.000, B 0.000, C 0.000 }
gfCNCPoint5[28690] = {X 258.1201, Y 51.9499, Z -8.0000, A 0.000, B 0.000, C 0.000 }
gfCNCPoint5[28691] = {X 257.0983, Y 51.5442, Z -8.0000, A 0.000, B 0.000, C 0.000 }
gfCNCPoint5[28692] = {X 256.1493, Y 50.9894, Z -8.0000, A 0.000, B 0.000, C 0.000 }
gfCNCPoint5[28693] = {X 255.2946, Y 50.2979, Z -8.0000, A 0.000, B 0.000, C 0.000 }
gfCNCPoint5[28694] = {X 255.1775, Y 50.1851, Z -8.0000, A 0.000, B 0.000, C 0.000 }
gfCNCPoint5[28695] = {X 255.0630, Y 50.0697, Z -8.0000, A 0.000, B 0.000, C 0.000 }
gfCNCPoint5[28696] = {X 254.3405, Y 49.1989, Z -8.0000, A 0.000, B 0.000, C 0.000 }
gfCNCPoint5[28697] = {X 253.7617, Y 48.2267, Z -8.0000, A 0.000, B 0.000, C 0.000 }
gfCNCPoint5[28698] = {X 253.3406, Y 47.1766, Z -8.0000, A 0.000, B 0.000, C 0.000 }
gfCNCPoint5[28699] = {X 252.9194, Y 48.2267, Z -8.0000, A 0.000, B 0.000, C 0.000 }
gfCNCPoint5[28700] = {X 252.3406, Y 49.1989, Z -8.0000, A 0.000, B 0.000, C 0.000 }
gfCNCPoint5[28701] = {X 251.6182, Y 50.0697, Z -8.0000, A 0.000, B 0.000, C 0.000 }
gfCNCPoint5[28702] = {X 251.5700, Y 50.1189, Z -8.0000, A 0.000, B 0.000, C 0.000 }
gfCNCPoint5[28703] = {X 251.5214, Y 50.1676, Z -8.0000, A 0.000, B 0.000, C 0.000 }
gfCNCPoint5[28704] = {X 250.7154, Y 50.8583, Z -8.0000, A 0.000, B 0.000, C 0.000 }
gfCNCPoint5[28705] = {X 249.8175, Y 51.4245, Z -8.0000, A 0.000, B 0.000, C 0.000 }
gfCNCPoint5[28706] = {X 248.8469, Y 51.8542, Z -8.0000, A 0.000, B 0.000, C 0.000 }
gfCNCPoint5[28707] = {X 247.8241, Y 52.1381, Z -8.0000, A 0.000, B 0.000, C 0.000 }
gfCNCPoint5[28708] = {X 247.8927, Y 52.2634, Z -8.0000, A 0.000, B 0.000, C 0.000 }
gfCNCPoint5[28709] = {X 247.9598, Y 52.3896, Z -8.0000, A 0.000, B 0.000, C 0.000 }
gfCNCPoint5[28710] = {X 250.9686, Y 53.5630, Z -8.0000, A 0.000, B 0.000, C 0.000 }
gfCNCPoint5[28711] = {X 252.7631, Y 54.2752, Z -8.0000, A 0.000, B 0.000, C 0.000 }
gfCNCPoint5[28712] = {X 251.8777, Y 56.5059, Z -8.0000, A 0.000, B 0.000, C 0.000 }
gfCNCPoint5[28713] = {X 267.2820, Y 62.6202, Z -8.0000, A 0.000, B 0.000, C 0.000 }
gfCNCPoint5[28714] = {X 266.8842, Y 61.4457, Z -8.0000, A 0.000, B 0.000, C 0.000 }
gfCNCPoint5[28715] = {X 266.6398, Y 60.2300, Z -8.0000, A 0.000, B 0.000, C 0.000 }
gfCNCPoint5[28716] = {X 266.5529, Y 58.9930, Z -8.0000, A 0.000, B 0.000, C 0.000 }
gfCNCPoint5[28717] = {X 266.5527, Y 58.0000, Z -8.0000, A 0.000, B 0.000, C 0.000 }
gfCNCPoint5[28718] = {X 266.6262, Y 56.8093, Z -8.0000, A 0.000, B 0.000, C 0.000 }
gfCNCPoint5[28719] = {X 266.8456, Y 55.6367, Z -8.0000, A 0.000, B 0.000, C 0.000 }
gfCNCPoint5[28720] = {X 267.2076, Y 54.5000, Z -8.0000, A 0.000, B 0.000, C 0.000 }
gfCNCPoint5[28721] = {X 267.7067, Y 53.4164, Z -8.0000, A 0.000, B 0.000, C 0.000 }
gfCNCPoint5[28722] = {X 268.4728, Y 52.2132, Z -8.0000, A 0.000, B 0.000, C 0.000 }
gfCNCPoint5[28723] = {X 269.4075, Y 51.1357, Z -8.0000, A 0.000, B 0.000, C 0.000 }
gfCNCPoint5[28724] = {X 270.4903, Y 50.2072, Z -8.0000, A 0.000, B 0.000, C 0.000 }
gfCNCPoint5[28725] = {X 271.6979, Y 49.4479, Z -8.0000, A 0.000, B 0.000, C 0.000 }
gfCNCPoint5[28726] = {X 273.0039, Y 48.8744, Z -8.0000, A 0.000, B 0.000, C 0.000 }
gfCNCPoint5[28727] = {X 274.3800, Y 48.4989, Z -8.0000, A 0.000, B 0.000, C 0.000 }
gfCNCPoint5[28728] = {X 275.3020, Y 48.3648, Z -8.0000, A 0.000, B 0.000, C 0.000 }
gfCNCPoint5[28729] = {X 276.2327, Y 48.3200, Z -8.0000, A 0.000, B 0.000, C 0.000 }
gfCNCPoint5[28730] = {X 281.0411, Y 48.3200, Z -8.0000, A 0.000, B 0.000, C 0.000 }
gfCNCPoint5[28731] = {X 280.4347, Y 47.5134, Z -8.0000, A 0.000, B 0.000, C 0.000 }
gfCNCPoint5[28732] = {X 280.0072, Y 46.5992, Z -8.0000, A 0.000, B 0.000, C 0.000 }
gfCNCPoint5[28733] = {X 279.7768, Y 45.6167, Z -8.0000, A 0.000, B 0.000, C 0.000 }
gfCNCPoint5[28734] = {X 279.7488, Y 45.3288, Z -8.0000, A 0.000, B 0.000, C 0.000 }
gfCNCPoint5[28735] = {X 279.7378, Y 45.0398, Z -8.0000, A 0.000, B 0.000, C 0.000 }
gfCNCPoint5[28736] = {X 279.7377, Y 44.2052, Z -8.0000, A 0.000, B 0.000, C 0.000 }
gfCNCPoint5[28737] = {X 279.8412, Y 43.2212, Z -8.0000, A 0.000, B 0.000, C 0.000 }
gfCNCPoint5[28738] = {X 280.1393, Y 42.2777, Z -8.0000, A 0.000, B 0.000, C 0.000 }
gfCNCPoint5[28739] = {X 280.6201, Y 41.4129, Z -8.0000, A 0.000, B 0.000, C 0.000 }
gfCNCPoint5[28740] = {X 281.2641, Y 40.6618, Z -8.0000, A 0.000, B 0.000, C 0.000 }
gfCNCPoint5[28741] = {X 281.2643, Y 16.5233, Z -8.0000, A 0.000, B 0.000, C 0.000 }
gfCNCPoint5[28742] = {X 280.6235, Y 15.7818, Z -8.0000, A 0.000, B 0.000, C 0.000 }
gfCNCPoint5[28743] = {X 280.1438, Y 14.9272, Z -8.0000, A 0.000, B 0.000, C 0.000 }
gfCNCPoint5[28744] = {X 279.8446, Y 13.9940, Z -8.0000, A 0.000, B 0.000, C 0.000 }
gfCNCPoint5[28745] = {X 279.7378, Y 13.0198, Z -8.0000, A 0.000, B 0.000, C 0.000 }
gfCNCPoint5[28746] = {X 279.7377, Y 12.1868, Z -8.0000, A 0.000, B 0.000, C 0.000 }
gfCNCPoint5[28747] = {X 279.8242, Y 11.2717, Z -8.0000, A 0.000, B 0.000, C 0.000 }
gfCNCPoint5[28748] = {X 280.0809, Y 10.3890, Z -8.0000, A 0.000, B 0.000, C 0.000 }
gfCNCPoint5[28749] = {X 280.5256, Y 9.5279, Z -8.0000, A 0.000, B 0.000, C 0.000 }
gfCNCPoint5[28750] = {X 281.1317, Y 8.7718, Z -8.0000, A 0.000, B 0.000, C 0.000 }
gfCNCPoint5[28751] = {X 281.8753, Y 8.1502, Z -8.0000, A 0.000, B 0.000, C 0.000 }
gfCNCPoint5[28752] = {X 282.7270, Y 7.6879, Z -8.0000, A 0.000, B 0.000, C 0.000 }
gfCNCPoint5[28753] = {X 283.6533, Y 7.4030, Z -8.0000, A 0.000, B 0.000, C 0.000 }
gfCNCPoint5[28754] = {X 284.6177, Y 7.3068, Z -8.0000, A 0.000, B 0.000, C 0.000 }
gfCNCPoint5[28755] = {X 291.0611, Y 7.3068, Z -8.0000, A 0.000, B 0.000, C 0.000 }
gfCNCPoint5[28756] = {X 292.0255, Y 7.4030, Z -8.0000, A 0.000, B 0.000, C 0.000 }
gfCNCPoint5[28757] = {X 292.9518, Y 7.6879, Z -8.0000, A 0.000, B 0.000, C 0.000 }
gfCNCPoint5[28758] = {X 293.8035, Y 8.1502, Z -8.0000, A 0.000, B 0.000, C 0.000 }
gfCNCPoint5[28759] = {X 294.5471, Y 8.7718, Z -8.0000, A 0.000, B 0.000, C 0.000 }
gfCNCPoint5[28760] = {X 295.1532, Y 9.5279, Z -8.0000, A 0.000, B 0.000, C 0.000 }
gfCNCPoint5[28761] = {X 295.5979, Y 10.3890, Z -8.0000, A 0.000, B 0.000, C 0.000 }
